LIN {X 0,Y 516.769,Z 315.126,A -85,B 0,C 180,E1 -4914.686,E2 -4914.686} C_VEL
LIN {X 0,Y 516.792,Z 318.611,A -85,B 0,C 180,E1 -4917.047,E2 -4917.047} C_VEL
LIN {X 0,Y 516.703,Z 322.745,A -85,B 0,C 180,E1 -4919.785,E2 -4919.785} C_VEL
LIN {X 0,Y 516.62,Z 326.844,A -85,B 0,C 180,E1 -4922.451,E2 -4922.451} C_VEL
LIN {X 0,Y 516.569,Z 330.921,A -85,B 0,C 180,E1 -4925.055,E2 -4925.055} C_VEL
LIN {X 0,Y 516.482,Z 335.169,A -85,B 0,C 180,E1 -4927.715,E2 -4927.715} C_VEL
LIN {X 0,Y 516.394,Z 340.454,A -85,B 0,C 180,E1 -4930.936,E2 -4930.936} C_VEL
LIN {X 0,Y 516.331,Z 344.572,A -85,B 0,C 180,E1 -4933.392,E2 -4933.392} C_VEL
LIN {X 0,Y 516.365,Z 349.185,A -85,B 0,C 180,E1 -4936.121,E2 -4936.121} C_VEL
LIN {X 0,Y 516.368,Z 349.452,A -85,B 0,C 180,E1 -4936.184,E2 -4936.184} C_VEL
LIN {X 0,Y 518.473,Z 361.595,A -85,B 0,C 180,E1 -4936.553,E2 -4936.553} C_VEL
LIN {X 0,Y 518.217,Z 374.075,A -85,B 0,C 180,E1 -4937.02,E2 -4937.02} C_VEL
LIN {X 0,Y 517.915,Z 385.417,A -85,B 0,C 180,E1 -4937.593,E2 -4937.593} C_VEL
LIN {X 0,Y 517.665,Z 396.987,A -85,B 0,C 180,E1 -4938.35,E2 -4938.35} C_VEL
LIN {X 0,Y 517.369,Z 407.679,A -85,B 0,C 180,E1 -4939.236,E2 -4939.236} C_VEL
LIN {X 0,Y 517.06,Z 417.299,A -85,B 0,C 180,E1 -4940.218,E2 -4940.218} C_VEL
LIN {X 0,Y 516.853,Z 425.177,A -85,B 0,C 180,E1 -4941.201,E2 -4941.201} C_VEL
LIN {X 0,Y 516.613,Z 432.881,A -85,B 0,C 180,E1 -4942.378,E2 -4942.378} C_VEL
LIN {X 0,Y 516.468,Z 439.944,A -85,B 0,C 180,E1 -4943.751,E2 -4943.751} C_VEL
LIN {X 0,Y 516.313,Z 444.654,A -85,B 0,C 180,E1 -4944.924,E2 -4944.924} C_VEL
LIN {X 0,Y 516.373,Z 448.256,A -85,B 0,C 180,E1 -4946.098,E2 -4946.098} C_VEL
LIN {X 0,Y 516.282,Z 450.122,A -85,B 0,C 180,E1 -4946.879,E2 -4946.879} C_VEL
LIN {X 0,Y 516.262,Z 451.529,A -85,B 0,C 180,E1 -4947.66,E2 -4947.66} C_VEL
LIN {X 0,Y 516.16,Z 453.147,A -85,B 0,C 180,E1 -4949.22,E2 -4949.22} C_VEL
LIN {X 0,Y 516.155,Z 453.384,A -85,B 0,C 180,E1 -4950,E2 -4950} C_VEL
LIN {X 0,Y 516.16,Z 453.201,A -85,B 0,C 180,E1 -4950.78,E2 -4950.78} C_VEL
LIN {X 0,Y 516.262,Z 451.653,A -85,B 0,C 180,E1 -4952.341,E2 -4952.341} C_VEL
LIN {X 0,Y 516.283,Z 450.3,A -85,B 0,C 180,E1 -4953.122,E2 -4953.122} C_VEL
LIN {X 0,Y 516.362,Z 447.439,A -85,B 0,C 180,E1 -4954.293,E2 -4954.293} C_VEL
LIN {X 0,Y 516.404,Z 443.561,A -85,B 0,C 180,E1 -4955.467,E2 -4955.467} C_VEL
LIN {X 0,Y 516.491,Z 437.713,A -85,B 0,C 180,E1 -4956.814,E2 -4956.814} C_VEL
LIN {X 0,Y 516.667,Z 431.036,A -85,B 0,C 180,E1 -4958.015,E2 -4958.015} C_VEL
LIN {X 0,Y 516.872,Z 422.892,A -85,B 0,C 180,E1 -4959.194,E2 -4959.194} C_VEL
LIN {X 0,Y 517.116,Z 414.554,A -85,B 0,C 180,E1 -4960.177,E2 -4960.177} C_VEL
LIN {X 0,Y 517.451,Z 404.26,A -85,B 0,C 180,E1 -4961.16,E2 -4961.16} C_VEL
LIN {X 0,Y 517.728,Z 393.047,A -85,B 0,C 180,E1 -4962.018,E2 -4962.018} C_VEL
LIN {X 0,Y 517.966,Z 382.905,A -85,B 0,C 180,E1 -4962.638,E2 -4962.638} C_VEL
LIN {X 0,Y 518.356,Z 370.372,A -85,B 0,C 180,E1 -4963.226,E2 -4963.226} C_VEL
LIN {X 0,Y 518.325,Z 360.107,A -85,B 0,C 180,E1 -4963.589,E2 -4963.589} C_VEL
LIN {X 0,Y 516.374,Z 349.251,A -85,B 0,C 180,E1 -4963.93,E2 -4963.93} C_VEL
LIN {X 0,Y 516.317,Z 344.726,A -85,B 0,C 180,E1 -4966.61,E2 -4966.61} C_VEL
LIN {X 0,Y 516.386,Z 340.608,A -85,B 0,C 180,E1 -4969.065,E2 -4969.065} C_VEL
LIN {X 0,Y 516.483,Z 335.316,A -85,B 0,C 180,E1 -4972.285,E2 -4972.285} C_VEL
LIN {X 0,Y 516.554,Z 331.064,A -85,B 0,C 180,E1 -4974.946,E2 -4974.946} C_VEL
LIN {X 0,Y 516.636,Z 326.528,A -85,B 0,C 180,E1 -4977.844,E2 -4977.844} C_VEL
LIN {X 0,Y 516.679,Z 322.893,A -85,B 0,C 180,E1 -4980.217,E2 -4980.217} C_VEL
LIN {X 0,Y 516.794,Z 318.755,A -85,B 0,C 180,E1 -4982.954,E2 -4982.954} C_VEL
LIN {X 0,Y 516.804,Z 315.253,A -85,B 0,C 180,E1 -4985.319,E2 -4985.319} C_VEL
LIN {X 0,Y 516.878,Z 315.1,A -85,B 0,C 180,E1 -4987.942,E2 -4987.942} C_VEL
LIN {X 0,Y 516.884,Z 315.101,A -85,B 0,C 180,E1 -4990.741,E2 -4990.741} C_VEL
LIN {X 0,Y 516.883,Z 315.098,A -85,B 0,C 180,E1 -4992.831,E2 -4992.831} C_VEL
LIN {X 0,Y 516.894,Z 315.096,A -85,B 0,C 180,E1 -4995.006,E2 -4995.006} C_VEL
LIN {X 0,Y 516.853,Z 315.103,A -85,B 0,C 180,E1 -4998.406,E2 -4998.406} C_VEL
LIN {X 0,Y 516.874,Z 315.1,A -85,B 0,C 180,E1 -5001.283,E2 -5001.283} C_VEL
LIN {X 0,Y 516.887,Z 315.101,A -85,B 0,C 180,E1 -5004.221,E2 -5004.221} C_VEL
LIN {X 0,Y 516.893,Z 315.098,A -85,B 0,C 180,E1 -5007.053,E2 -5007.053} C_VEL
LIN {X 0,Y 516.863,Z 315.1,A -85,B 0,C 180,E1 -5009.794,E2 -5009.794} C_VEL
LIN {X 0,Y 516.871,Z 315.102,A -85,B 0,C 180,E1 -5012.464,E2 -5012.464} C_VEL
LIN {X 0,Y 516.846,Z 315.104,A -85,B 0,C 180,E1 -5015.068,E2 -5015.068} C_VEL
LIN {X 0,Y 516.864,Z 315.105,A -85,B 0,C 180,E1 -5017.621,E2 -5017.621} C_VEL
LIN {X 0,Y 516.928,Z 315.093,A -85,B 0,C 180,E1 -5020.13,E2 -5020.13} C_VEL
LIN {X 0,Y 516.915,Z 315.096,A -85,B 0,C 180,E1 -5022.596,E2 -5022.596} C_VEL
LIN {X 0,Y 516.934,Z 315.093,A -85,B 0,C 180,E1 -5025.03,E2 -5025.03} C_VEL
LIN {X 0,Y 516.961,Z 315.094,A -85,B 0,C 180,E1 -5028.233,E2 -5028.233} C_VEL
LIN {X 0,Y 516.964,Z 315.092,A -85,B 0,C 180,E1 -5031.4,E2 -5031.4} C_VEL
LIN {X 0,Y 517.012,Z 315.083,A -85,B 0,C 180,E1 -5033.757,E2 -5033.757} C_VEL
LIN {X 0,Y 517.079,Z 315.073,A -85,B 0,C 180,E1 -5037.663,E2 -5037.663} C_VEL
LIN {X 0,Y 517.038,Z 315.079,A -85,B 0,C 180,E1 -5040.779,E2 -5040.779} C_VEL
LIN {X 0,Y 517.004,Z 315.086,A -85,B 0,C 180,E1 -5043.117,E2 -5043.117} C_VEL
LIN {X 0,Y 517.012,Z 315.083,A -85,B 0,C 180,E1 -5046.243,E2 -5046.243} C_VEL
LIN {X 0,Y 516.95,Z 315.089,A -85,B 0,C 180,E1 -5049.389,E2 -5049.389} C_VEL
LIN {X 0,Y 516.946,Z 315.093,A -85,B 0,C 180,E1 -5051.807,E2 -5051.807} C_VEL
LIN {X 0,Y 516.93,Z 315.094,A -85,B 0,C 180,E1 -5055.143,E2 -5055.143} C_VEL
LIN {X 0,Y 516.92,Z 315.095,A -85,B 0,C 180,E1 -5058.222,E2 -5058.222} C_VEL
LIN {X 0,Y 516.909,Z 315.098,A -85,B 0,C 180,E1 -5060.702,E2 -5060.702} C_VEL
LIN {X 0,Y 516.868,Z 315.1,A -85,B 0,C 180,E1 -5063.224,E2 -5063.224} C_VEL
LIN {X 0,Y 516.893,Z 315.097,A -85,B 0,C 180,E1 -5066.186,E2 -5066.186} C_VEL
LIN {X 0,Y 516.881,Z 315.101,A -85,B 0,C 180,E1 -5069.519,E2 -5069.519} C_VEL
LIN {X 0,Y 516.894,Z 315.1,A -85,B 0,C 180,E1 -5072.544,E2 -5072.544} C_VEL
LIN {X 0,Y 516.878,Z 315.1,A -85,B 0,C 180,E1 -5075.332,E2 -5075.332} C_VEL
LIN {X 0,Y 516.877,Z 315.101,A -85,B 0,C 180,E1 -5077.943,E2 -5077.943} C_VEL
LIN {X 0,Y 516.849,Z 315.103,A -85,B 0,C 180,E1 -5080.745,E2 -5080.745} C_VEL
LIN {X 0,Y 516.878,Z 315.099,A -85,B 0,C 180,E1 -5083.904,E2 -5083.904} C_VEL
LIN {X 0,Y 516.88,Z 315.103,A -85,B 0,C 180,E1 -5086.107,E2 -5086.107} C_VEL
LIN {X 0,Y 516.915,Z 315.097,A -85,B 0,C 180,E1 -5088.399,E2 -5088.399} C_VEL
LIN {X 0,Y 516.88,Z 315.104,A -85,B 0,C 180,E1 -5091.284,E2 -5091.284} C_VEL
LIN {X 0,Y 516.893,Z 315.205,A -85,B 0,C 180,E1 -5092.277,E2 -5092.277} C_VEL
LIN {X 0,Y 517.584,Z 320.371,A -85,B 0,C 180,E1 -5094.559,E2 -5094.559} C_VEL
LIN {X 0,Y 517.453,Z 327.148,A -85,B 0,C 180,E1 -5097.361,E2 -5097.361} C_VEL
LIN {X 0,Y 517.277,Z 334.775,A -85,B 0,C 180,E1 -5100.405,E2 -5100.405} C_VEL
LIN {X 0,Y 517.083,Z 342.335,A -85,B 0,C 180,E1 -5103.351,E2 -5103.351} C_VEL
LIN {X 0,Y 516.938,Z 350.126,A -85,B 0,C 180,E1 -5106.355,E2 -5106.355} C_VEL
LIN {X 0,Y 516.789,Z 357.918,A -85,B 0,C 180,E1 -5109.293,E2 -5109.293} C_VEL
LIN {X 0,Y 516.635,Z 365.829,A -85,B 0,C 180,E1 -5112.221,E2 -5112.221} C_VEL
LIN {X 0,Y 516.567,Z 373.5,A -85,B 0,C 180,E1 -5115.019,E2 -5115.019} C_VEL
LIN {X 0,Y 516.505,Z 376.491,A -85,B 0,C 180,E1 -5116.099,E2 -5116.099} C_VEL
LIN {X 0,Y 518.478,Z 389.092,A -85,B 0,C 180,E1 -5116.453,E2 -5116.453} C_VEL
LIN {X 0,Y 518.244,Z 402.111,A -85,B 0,C 180,E1 -5116.92,E2 -5116.92} C_VEL
LIN {X 0,Y 517.912,Z 414.402,A -85,B 0,C 180,E1 -5117.529,E2 -5117.529} C_VEL
LIN {X 0,Y 517.617,Z 425.586,A -85,B 0,C 180,E1 -5118.249,E2 -5118.249} C_VEL
LIN {X 0,Y 517.328,Z 436.469,A -85,B 0,C 180,E1 -5119.135,E2 -5119.135} C_VEL
LIN {X 0,Y 517.044,Z 445.333,A -85,B 0,C 180,E1 -5120.02,E2 -5120.02} C_VEL
LIN {X 0,Y 516.814,Z 454.959,A -85,B 0,C 180,E1 -5121.2,E2 -5121.2} C_VEL
LIN {X 0,Y 516.563,Z 462.62,A -85,B 0,C 180,E1 -5122.377,E2 -5122.377} C_VEL
LIN {X 0,Y 516.427,Z 469.679,A -85,B 0,C 180,E1 -5123.75,E2 -5123.75} C_VEL
LIN {X 0,Y 516.313,Z 474.372,A -85,B 0,C 180,E1 -5124.924,E2 -5124.924} C_VEL
LIN {X 0,Y 516.355,Z 477.957,A -85,B 0,C 180,E1 -5126.098,E2 -5126.098} C_VEL
LIN {X 0,Y 516.282,Z 479.807,A -85,B 0,C 180,E1 -5126.878,E2 -5126.878} C_VEL
LIN {X 0,Y 516.261,Z 481.196,A -85,B 0,C 180,E1 -5127.659,E2 -5127.659} C_VEL
LIN {X 0,Y 516.16,Z 482.785,A -85,B 0,C 180,E1 -5129.22,E2 -5129.22} C_VEL
LIN {X 0,Y 516.154,Z 483,A -85,B 0,C 180,E1 -5130,E2 -5130} C_VEL
LIN {X 0,Y 516.192,Z 482.186,A -85,B 0,C 180,E1 -5131.56,E2 -5131.56} C_VEL
LIN {X 0,Y 516.261,Z 481.199,A -85,B 0,C 180,E1 -5132.34,E2 -5132.34} C_VEL
LIN {X 0,Y 516.282,Z 479.811,A -85,B 0,C 180,E1 -5133.121,E2 -5133.121} C_VEL
LIN {X 0,Y 516.343,Z 476.897,A -85,B 0,C 180,E1 -5134.293,E2 -5134.293} C_VEL
LIN {X 0,Y 516.405,Z 472.95,A -85,B 0,C 180,E1 -5135.466,E2 -5135.466} C_VEL
LIN {X 0,Y 516.485,Z 467.035,A -85,B 0,C 180,E1 -5136.807,E2 -5136.807} C_VEL
LIN {X 0,Y 516.64,Z 460.24,A -85,B 0,C 180,E1 -5138.015,E2 -5138.015} C_VEL
LIN {X 0,Y 516.867,Z 451.995,A -85,B 0,C 180,E1 -5139.193,E2 -5139.193} C_VEL
LIN {X 0,Y 517.08,Z 443.544,A -85,B 0,C 180,E1 -5140.177,E2 -5140.177} C_VEL
LIN {X 0,Y 517.46,Z 433.103,A -85,B 0,C 180,E1 -5141.159,E2 -5141.159} C_VEL
LIN {X 0,Y 517.696,Z 421.809,A -85,B 0,C 180,E1 -5142.014,E2 -5142.014} C_VEL
LIN {X 0,Y 517.97,Z 411.419,A -85,B 0,C 180,E1 -5142.637,E2 -5142.637} C_VEL
LIN {X 0,Y 518.28,Z 399.779,A -85,B 0,C 180,E1 -5143.178,E2 -5143.178} C_VEL
LIN {X 0,Y 518.314,Z 387.284,A -85,B 0,C 180,E1 -5143.601,E2 -5143.601} C_VEL
LIN {X 0,Y 516.504,Z 376.493,A -85,B 0,C 180,E1 -5143.9,E2 -5143.9} C_VEL
LIN {X 0,Y 516.576,Z 369.05,A -85,B 0,C 180,E1 -5146.6,E2 -5146.6} C_VEL
LIN {X 0,Y 516.77,Z 360.146,A -85,B 0,C 180,E1 -5149.876,E2 -5149.876} C_VEL
LIN {X 0,Y 516.909,Z 352.356,A -85,B 0,C 180,E1 -5152.797,E2 -5152.797} C_VEL
LIN {X 0,Y 517.036,Z 344.563,A -85,B 0,C 180,E1 -5155.783,E2 -5155.783} C_VEL
LIN {X 0,Y 517.178,Z 337.818,A -85,B 0,C 180,E1 -5158.399,E2 -5158.399} C_VEL
LIN {X 0,Y 517.364,Z 330.793,A -85,B 0,C 180,E1 -5161.151,E2 -5161.151} C_VEL
LIN {X 0,Y 517.541,Z 323.649,A -85,B 0,C 180,E1 -5164.07,E2 -5164.07} C_VEL
LIN {X 0,Y 517.565,Z 319.707,A -85,B 0,C 180,E1 -5165.724,E2 -5165.724} C_VEL
LIN {X 0,Y 516.89,Z 315.102,A -85,B 0,C 180,E1 -5167.8,E2 -5167.8} C_VEL
LIN {X 0,Y 516.9,Z 315.1,A -85,B 0,C 180,E1 -5170.739,E2 -5170.739} C_VEL
LIN {X 0,Y 516.878,Z 315.105,A -85,B 0,C 180,E1 -5173.902,E2 -5173.902} C_VEL
LIN {X 0,Y 516.875,Z 315.099,A -85,B 0,C 180,E1 -5176.106,E2 -5176.106} C_VEL
LIN {X 0,Y 516.853,Z 315.102,A -85,B 0,C 180,E1 -5179.255,E2 -5179.255} C_VEL
LIN {X 0,Y 516.873,Z 315.101,A -85,B 0,C 180,E1 -5182.056,E2 -5182.056} C_VEL
LIN {X 0,Y 516.887,Z 315.099,A -85,B 0,C 180,E1 -5185.175,E2 -5185.175} C_VEL
LIN {X 0,Y 516.867,Z 315.102,A -85,B 0,C 180,E1 -5187.975,E2 -5187.975} C_VEL
LIN {X 0,Y 516.893,Z 315.102,A -85,B 0,C 180,E1 -5190.694,E2 -5190.694} C_VEL
LIN {X 0,Y 516.893,Z 315.097,A -85,B 0,C 180,E1 -5193.812,E2 -5193.812} C_VEL
LIN {X 0,Y 516.862,Z 315.101,A -85,B 0,C 180,E1 -5196.776,E2 -5196.776} C_VEL
LIN {X 0,Y 516.93,Z 315.096,A -85,B 0,C 180,E1 -5199.731,E2 -5199.731} C_VEL
LIN {X 0,Y 516.916,Z 315.098,A -85,B 0,C 180,E1 -5202.596,E2 -5202.596} C_VEL
LIN {X 0,Y 516.923,Z 315.094,A -85,B 0,C 180,E1 -5205.03,E2 -5205.03} C_VEL
LIN {X 0,Y 516.955,Z 315.092,A -85,B 0,C 180,E1 -5208.233,E2 -5208.233} C_VEL
LIN {X 0,Y 516.962,Z 315.092,A -85,B 0,C 180,E1 -5211.4,E2 -5211.4} C_VEL
LIN {X 0,Y 517.053,Z 315.08,A -85,B 0,C 180,E1 -5214.54,E2 -5214.54} C_VEL
LIN {X 0,Y 517.074,Z 315.075,A -85,B 0,C 180,E1 -5217.663,E2 -5217.663} C_VEL
LIN {X 0,Y 517.053,Z 315.076,A -85,B 0,C 180,E1 -5220.779,E2 -5220.779} C_VEL
LIN {X 0,Y 517.001,Z 315.085,A -85,B 0,C 180,E1 -5223.117,E2 -5223.117} C_VEL
LIN {X 0,Y 517.007,Z 315.083,A -85,B 0,C 180,E1 -5226.243,E2 -5226.243} C_VEL
LIN {X 0,Y 516.946,Z 315.091,A -85,B 0,C 180,E1 -5229.389,E2 -5229.389} C_VEL
LIN {X 0,Y 516.94,Z 315.096,A -85,B 0,C 180,E1 -5231.807,E2 -5231.807} C_VEL
LIN {X 0,Y 516.927,Z 315.095,A -85,B 0,C 180,E1 -5235.144,E2 -5235.144} C_VEL
LIN {X 0,Y 516.916,Z 315.094,A -85,B 0,C 180,E1 -5238.223,E2 -5238.223} C_VEL
LIN {X 0,Y 516.904,Z 315.101,A -85,B 0,C 180,E1 -5240.702,E2 -5240.702} C_VEL
LIN {X 0,Y 516.863,Z 315.101,A -85,B 0,C 180,E1 -5243.224,E2 -5243.224} C_VEL
LIN {X 0,Y 516.893,Z 315.099,A -85,B 0,C 180,E1 -5246.188,E2 -5246.188} C_VEL
LIN {X 0,Y 516.876,Z 315.1,A -85,B 0,C 180,E1 -5249.519,E2 -5249.519} C_VEL
LIN {X 0,Y 516.89,Z 315.102,A -85,B 0,C 180,E1 -5252.545,E2 -5252.545} C_VEL
LIN {X 0,Y 516.876,Z 315.1,A -85,B 0,C 180,E1 -5255.333,E2 -5255.333} C_VEL
LIN {X 0,Y 516.873,Z 315.103,A -85,B 0,C 180,E1 -5257.944,E2 -5257.944} C_VEL
LIN {X 0,Y 516.854,Z 315.104,A -85,B 0,C 180,E1 -5260.745,E2 -5260.745} C_VEL
LIN {X 0,Y 516.875,Z 315.099,A -85,B 0,C 180,E1 -5263.904,E2 -5263.904} C_VEL
LIN {X 0,Y 516.863,Z 315.099,A -85,B 0,C 180,E1 -5266.924,E2 -5266.924} C_VEL
LIN {X 0,Y 516.905,Z 315.098,A -85,B 0,C 180,E1 -5269.588,E2 -5269.588} C_VEL
LIN {X 0,Y 516.898,Z 315.097,A -85,B 0,C 180,E1 -5270.31,E2 -5270.31} C_VEL
LIN {X 0,Y 516.218,Z 315.184,A -85,B 0,C 180,E1 -5270.96,E2 -5270.96} C_VEL
LIN {X 0,Y 513.359,Z 315.539,A -85,B 0,C 180,E1 -5272.015,E2 -5272.015} C_VEL
LIN {X 0,Y 510.934,Z 315.843,A -85,B 0,C 180,E1 -5272.865,E2 -5272.865} C_VEL
LIN {X 0,Y 509.869,Z 315.975,A -85,B 0,C 180,E1 -5273.522,E2 -5273.522} C_VEL
LIN {X 0,Y 509.769,Z 315.986,A -85,B 0,C 180,E1 -5273.744,E2 -5273.744} C_VEL
LIN {X 0,Y 509.741,Z 315.993,A -85,B 0,C 180,E1 -5274.616,E2 -5274.616} C_VEL
LIN {X 0,Y 509.762,Z 318.703,A -85,B 0,C 180,E1 -5276.533,E2 -5276.533} C_VEL
LIN {X 0,Y 509.647,Z 322.848,A -85,B 0,C 180,E1 -5279.322,E2 -5279.322} C_VEL
LIN {X 0,Y 509.592,Z 326.962,A -85,B 0,C 180,E1 -5282.038,E2 -5282.038} C_VEL
LIN {X 0,Y 509.535,Z 332.407,A -85,B 0,C 180,E1 -5285.558,E2 -5285.558} C_VEL
LIN {X 0,Y 509.372,Z 336.479,A -85,B 0,C 180,E1 -5288.129,E2 -5288.129} C_VEL
LIN {X 0,Y 509.318,Z 340.577,A -85,B 0,C 180,E1 -5290.661,E2 -5290.661} C_VEL
LIN {X 0,Y 509.269,Z 344.729,A -85,B 0,C 180,E1 -5293.155,E2 -5293.155} C_VEL
LIN {X 0,Y 509.311,Z 349.492,A -85,B 0,C 180,E1 -5295.976,E2 -5295.976} C_VEL
LIN {X 0,Y 511.573,Z 362.589,A -85,B 0,C 180,E1 -5296.393,E2 -5296.393} C_VEL
LIN {X 0,Y 511.276,Z 375.432,A -85,B 0,C 180,E1 -5296.891,E2 -5296.891} C_VEL
LIN {X 0,Y 510.976,Z 387.064,A -85,B 0,C 180,E1 -5297.504,E2 -5297.504} C_VEL
LIN {X 0,Y 510.698,Z 398.496,A -85,B 0,C 180,E1 -5298.289,E2 -5298.289} C_VEL
LIN {X 0,Y 510.363,Z 408.966,A -85,B 0,C 180,E1 -5299.186,E2 -5299.186} C_VEL
LIN {X 0,Y 510.066,Z 417.52,A -85,B 0,C 180,E1 -5300.083,E2 -5300.083} C_VEL
LIN {X 0,Y 509.836,Z 425.397,A -85,B 0,C 180,E1 -5301.079,E2 -5301.079} C_VEL
LIN {X 0,Y 509.569,Z 433.1,A -85,B 0,C 180,E1 -5302.272,E2 -5302.272} C_VEL
LIN {X 0,Y 509.403,Z 440.162,A -85,B 0,C 180,E1 -5303.664,E2 -5303.664} C_VEL
LIN {X 0,Y 509.248,Z 444.871,A -85,B 0,C 180,E1 -5304.854,E2 -5304.854} C_VEL
LIN {X 0,Y 509.303,Z 448.473,A -85,B 0,C 180,E1 -5306.044,E2 -5306.044} C_VEL
LIN {X 0,Y 509.201,Z 450.339,A -85,B 0,C 180,E1 -5306.836,E2 -5306.836} C_VEL
LIN {X 0,Y 509.19,Z 451.744,A -85,B 0,C 180,E1 -5307.627,E2 -5307.627} C_VEL
LIN {X 0,Y 509.074,Z 453.362,A -85,B 0,C 180,E1 -5309.209,E2 -5309.209} C_VEL
LIN {X 0,Y 509.066,Z 453.599,A -85,B 0,C 180,E1 -5310,E2 -5310} C_VEL
LIN {X 0,Y 509.074,Z 453.416,A -85,B 0,C 180,E1 -5310.791,E2 -5310.791} C_VEL
LIN {X 0,Y 509.19,Z 451.867,A -85,B 0,C 180,E1 -5312.373,E2 -5312.373} C_VEL
LIN {X 0,Y 509.202,Z 450.514,A -85,B 0,C 180,E1 -5313.165,E2 -5313.165} C_VEL
LIN {X 0,Y 509.284,Z 447.653,A -85,B 0,C 180,E1 -5314.353,E2 -5314.353} C_VEL
LIN {X 0,Y 509.347,Z 443.774,A -85,B 0,C 180,E1 -5315.543,E2 -5315.543} C_VEL
LIN {X 0,Y 509.419,Z 438.149,A -85,B 0,C 180,E1 -5316.865,E2 -5316.865} C_VEL
LIN {X 0,Y 509.63,Z 431.248,A -85,B 0,C 180,E1 -5318.126,E2 -5318.126} C_VEL
LIN {X 0,Y 509.86,Z 423.103,A -85,B 0,C 180,E1 -5319.321,E2 -5319.321} C_VEL
LIN {X 0,Y 510.118,Z 414.765,A -85,B 0,C 180,E1 -5320.318,E2 -5320.318} C_VEL
LIN {X 0,Y 510.498,Z 404.467,A -85,B 0,C 180,E1 -5321.314,E2 -5321.314} C_VEL
LIN {X 0,Y 510.781,Z 393.254,A -85,B 0,C 180,E1 -5322.184,E2 -5322.184} C_VEL
LIN {X 0,Y 511.038,Z 383.11,A -85,B 0,C 180,E1 -5322.812,E2 -5322.812} C_VEL
LIN {X 0,Y 511.466,Z 370.571,A -85,B 0,C 180,E1 -5323.408,E2 -5323.408} C_VEL
LIN {X 0,Y 511.377,Z 360.716,A -85,B 0,C 180,E1 -5323.765,E2 -5323.765} C_VEL
LIN {X 0,Y 509.3,Z 349.471,A -85,B 0,C 180,E1 -5324.127,E2 -5324.127} C_VEL
LIN {X 0,Y 509.255,Z 344.881,A -85,B 0,C 180,E1 -5326.847,E2 -5326.847} C_VEL
LIN {X 0,Y 509.313,Z 340.73,A -85,B 0,C 180,E1 -5329.34,E2 -5329.34} C_VEL
LIN {X 0,Y 509.425,Z 335.728,A -85,B 0,C 180,E1 -5332.432,E2 -5332.432} C_VEL
LIN {X 0,Y 509.492,Z 331.193,A -85,B 0,C 180,E1 -5335.316,E2 -5335.316} C_VEL
LIN {X 0,Y 509.572,Z 327,A -85,B 0,C 180,E1 -5338.031,E2 -5338.031} C_VEL
LIN {X 0,Y 509.655,Z 322.148,A -85,B 0,C 180,E1 -5341.244,E2 -5341.244} C_VEL
LIN {X 0,Y 509.812,Z 317.769,A -85,B 0,C 180,E1 -5344.195,E2 -5344.195} C_VEL
LIN {X 0,Y 509.767,Z 315.987,A -85,B 0,C 180,E1 -5345.569,E2 -5345.569} C_VEL
LIN {X 0,Y 509.848,Z 315.978,A -85,B 0,C 180,E1 -5348.338,E2 -5348.338} C_VEL
LIN {X 0,Y 509.857,Z 315.974,A -85,B 0,C 180,E1 -5351.425,E2 -5351.425} C_VEL
LIN {X 0,Y 509.838,Z 315.974,A -85,B 0,C 180,E1 -5354.669,E2 -5354.669} C_VEL
LIN {X 0,Y 509.789,Z 315.985,A -85,B 0,C 180,E1 -5357.505,E2 -5357.505} C_VEL
LIN {X 0,Y 509.83,Z 315.98,A -85,B 0,C 180,E1 -5360.646,E2 -5360.646} C_VEL
LIN {X 0,Y 509.832,Z 315.979,A -85,B 0,C 180,E1 -5363.647,E2 -5363.647} C_VEL
LIN {X 0,Y 509.859,Z 315.973,A -85,B 0,C 180,E1 -5366.539,E2 -5366.539} C_VEL
LIN {X 0,Y 509.831,Z 315.981,A -85,B 0,C 180,E1 -5369.333,E2 -5369.333} C_VEL
LIN {X 0,Y 509.827,Z 315.977,A -85,B 0,C 180,E1 -5372.05,E2 -5372.05} C_VEL
LIN {X 0,Y 509.802,Z 315.983,A -85,B 0,C 180,E1 -5374.7,E2 -5374.7} C_VEL
LIN {X 0,Y 509.822,Z 315.981,A -85,B 0,C 180,E1 -5377.458,E2 -5377.458} C_VEL
LIN {X 0,Y 509.913,Z 315.968,A -85,B 0,C 180,E1 -5379.844,E2 -5379.844} C_VEL
LIN {X 0,Y 509.874,Z 315.973,A -85,B 0,C 180,E1 -5383.174,E2 -5383.174} C_VEL
LIN {X 0,Y 509.847,Z 315.974,A -85,B 0,C 180,E1 -5385.634,E2 -5385.634} C_VEL
LIN {X 0,Y 509.907,Z 315.968,A -85,B 0,C 180,E1 -5388.874,E2 -5388.874} C_VEL
LIN {X 0,Y 509.947,Z 315.964,A -85,B 0,C 180,E1 -5392.078,E2 -5392.078} C_VEL
LIN {X 0,Y 509.982,Z 315.96,A -85,B 0,C 180,E1 -5394.464,E2 -5394.464} C_VEL
LIN {X 0,Y 510.049,Z 315.948,A -85,B 0,C 180,E1 -5397.631,E2 -5397.631} C_VEL
LIN {X 0,Y 509.99,Z 315.957,A -85,B 0,C 180,E1 -5400.79,E2 -5400.79} C_VEL
LIN {X 0,Y 509.946,Z 315.965,A -85,B 0,C 180,E1 -5403.16,E2 -5403.16} C_VEL
LIN {X 0,Y 509.979,Z 315.96,A -85,B 0,C 180,E1 -5406.33,E2 -5406.33} C_VEL
LIN {X 0,Y 509.913,Z 315.969,A -85,B 0,C 180,E1 -5408.72,E2 -5408.72} C_VEL
LIN {X 0,Y 509.898,Z 315.973,A -85,B 0,C 180,E1 -5411.932,E2 -5411.932} C_VEL
LIN {X 0,Y 509.889,Z 315.972,A -85,B 0,C 180,E1 -5415.242,E2 -5415.242} C_VEL
LIN {X 0,Y 509.862,Z 315.976,A -85,B 0,C 180,E1 -5418.484,E2 -5418.484} C_VEL
LIN {X 0,Y 509.847,Z 315.977,A -85,B 0,C 180,E1 -5421.002,E2 -5421.002} C_VEL
LIN {X 0,Y 509.826,Z 315.979,A -85,B 0,C 180,E1 -5423.564,E2 -5423.564} C_VEL
LIN {X 0,Y 509.849,Z 315.973,A -85,B 0,C 180,E1 -5426.366,E2 -5426.366} C_VEL
LIN {X 0,Y 509.848,Z 315.975,A -85,B 0,C 180,E1 -5429.725,E2 -5429.725} C_VEL
LIN {X 0,Y 509.871,Z 315.976,A -85,B 0,C 180,E1 -5432.775,E2 -5432.775} C_VEL
LIN {X 0,Y 509.838,Z 315.978,A -85,B 0,C 180,E1 -5435.581,E2 -5435.581} C_VEL
LIN {X 0,Y 509.846,Z 315.975,A -85,B 0,C 180,E1 -5438.339,E2 -5438.339} C_VEL
LIN {X 0,Y 509.804,Z 315.982,A -85,B 0,C 180,E1 -5441.431,E2 -5441.431} C_VEL
LIN {X 0,Y 509.837,Z 315.981,A -85,B 0,C 180,E1 -5444.67,E2 -5444.67} C_VEL
LIN {X 0,Y 509.857,Z 315.979,A -85,B 0,C 180,E1 -5448.104,E2 -5448.104} C_VEL
LIN {X 0,Y 509.845,Z 315.978,A -85,B 0,C 180,E1 -5450.648,E2 -5450.648} C_VEL
LIN {X 0,Y 509.881,Z 316.03,A -85,B 0,C 180,E1 -5452.072,E2 -5452.072} C_VEL
LIN {X 0,Y 510.556,Z 320.994,A -85,B 0,C 180,E1 -5454.308,E2 -5454.308} C_VEL
LIN {X 0,Y 510.523,Z 326.406,A -85,B 0,C 180,E1 -5456.589,E2 -5456.589} C_VEL
LIN {X 0,Y 510.308,Z 333.217,A -85,B 0,C 180,E1 -5459.365,E2 -5459.365} C_VEL
LIN {X 0,Y 510.169,Z 340.015,A -85,B 0,C 180,E1 -5462.071,E2 -5462.071} C_VEL
LIN {X 0,Y 510,Z 346.787,A -85,B 0,C 180,E1 -5464.711,E2 -5464.711} C_VEL
LIN {X 0,Y 509.854,Z 353.867,A -85,B 0,C 180,E1 -5467.451,E2 -5467.451} C_VEL
LIN {X 0,Y 509.654,Z 362.37,A -85,B 0,C 180,E1 -5470.673,E2 -5470.673} C_VEL
LIN {X 0,Y 509.517,Z 371.274,A -85,B 0,C 180,E1 -5473.986,E2 -5473.986} C_VEL
LIN {X 0,Y 509.444,Z 376.491,A -85,B 0,C 180,E1 -5475.902,E2 -5475.902} C_VEL
LIN {X 0,Y 511.563,Z 389.927,A -85,B 0,C 180,E1 -5476.291,E2 -5476.291} C_VEL
LIN {X 0,Y 511.342,Z 402.11,A -85,B 0,C 180,E1 -5476.741,E2 -5476.741} C_VEL
LIN {X 0,Y 510.992,Z 413.172,A -85,B 0,C 180,E1 -5477.287,E2 -5477.287} C_VEL
LIN {X 0,Y 510.741,Z 423.844,A -85,B 0,C 180,E1 -5477.964,E2 -5477.964} C_VEL
LIN {X 0,Y 510.429,Z 434.261,A -85,B 0,C 180,E1 -5478.785,E2 -5478.785} C_VEL
LIN {X 0,Y 510.07,Z 443.538,A -85,B 0,C 180,E1 -5479.681,E2 -5479.681} C_VEL
LIN {X 0,Y 509.846,Z 451.99,A -85,B 0,C 180,E1 -5480.679,E2 -5480.679} C_VEL
LIN {X 0,Y 509.585,Z 460.235,A -85,B 0,C 180,E1 -5481.873,E2 -5481.873} C_VEL
LIN {X 0,Y 509.419,Z 466.876,A -85,B 0,C 180,E1 -5483.067,E2 -5483.067} C_VEL
LIN {X 0,Y 509.344,Z 472.949,A -85,B 0,C 180,E1 -5484.457,E2 -5484.457} C_VEL
LIN {X 0,Y 509.234,Z 476.894,A -85,B 0,C 180,E1 -5485.646,E2 -5485.646} C_VEL
LIN {X 0,Y 509.201,Z 479.807,A -85,B 0,C 180,E1 -5486.835,E2 -5486.835} C_VEL
LIN {X 0,Y 509.161,Z 481.195,A -85,B 0,C 180,E1 -5487.626,E2 -5487.626} C_VEL
LIN {X 0,Y 509.073,Z 482.785,A -85,B 0,C 180,E1 -5489.209,E2 -5489.209} C_VEL
LIN {X 0,Y 509.065,Z 483,A -85,B 0,C 180,E1 -5490,E2 -5490} C_VEL
LIN {X 0,Y 509.112,Z 482.185,A -85,B 0,C 180,E1 -5491.582,E2 -5491.582} C_VEL
LIN {X 0,Y 509.161,Z 481.198,A -85,B 0,C 180,E1 -5492.373,E2 -5492.373} C_VEL
LIN {X 0,Y 509.2,Z 479.811,A -85,B 0,C 180,E1 -5493.164,E2 -5493.164} C_VEL
LIN {X 0,Y 509.234,Z 476.897,A -85,B 0,C 180,E1 -5494.353,E2 -5494.353} C_VEL
LIN {X 0,Y 509.344,Z 472.95,A -85,B 0,C 180,E1 -5495.542,E2 -5495.542} C_VEL
LIN {X 0,Y 509.409,Z 467.284,A -85,B 0,C 180,E1 -5496.853,E2 -5496.853} C_VEL
LIN {X 0,Y 509.584,Z 460.24,A -85,B 0,C 180,E1 -5498.126,E2 -5498.126} C_VEL
LIN {X 0,Y 509.845,Z 451.995,A -85,B 0,C 180,E1 -5499.321,E2 -5499.321} C_VEL
LIN {X 0,Y 510.069,Z 443.544,A -85,B 0,C 180,E1 -5500.318,E2 -5500.318} C_VEL
LIN {X 0,Y 510.486,Z 433.102,A -85,B 0,C 180,E1 -5501.313,E2 -5501.313} C_VEL
LIN {X 0,Y 510.729,Z 422.539,A -85,B 0,C 180,E1 -5502.129,E2 -5502.129} C_VEL
LIN {X 0,Y 511.037,Z 411.418,A -85,B 0,C 180,E1 -5502.812,E2 -5502.812} C_VEL
LIN {X 0,Y 511.374,Z 399.779,A -85,B 0,C 180,E1 -5503.359,E2 -5503.359} C_VEL
LIN {X 0,Y 511.411,Z 388.198,A -85,B 0,C 180,E1 -5503.763,E2 -5503.763} C_VEL
LIN {X 0,Y 509.443,Z 376.493,A -85,B 0,C 180,E1 -5504.097,E2 -5504.097} C_VEL
LIN {X 0,Y 509.522,Z 369.05,A -85,B 0,C 180,E1 -5506.837,E2 -5506.837} C_VEL
LIN {X 0,Y 509.711,Z 361.259,A -85,B 0,C 180,E1 -5509.743,E2 -5509.743} C_VEL
LIN {X 0,Y 509.85,Z 353.467,A -85,B 0,C 180,E1 -5512.703,E2 -5512.703} C_VEL
LIN {X 0,Y 510.001,Z 345.67,A -85,B 0,C 180,E1 -5515.726,E2 -5515.726} C_VEL
LIN {X 0,Y 510.18,Z 337.71,A -85,B 0,C 180,E1 -5518.824,E2 -5518.824} C_VEL
LIN {X 0,Y 510.375,Z 330.88,A -85,B 0,C 180,E1 -5521.551,E2 -5521.551} C_VEL
LIN {X 0,Y 510.547,Z 324.131,A -85,B 0,C 180,E1 -5524.359,E2 -5524.359} C_VEL
LIN {X 0,Y 510.453,Z 319.611,A -85,B 0,C 180,E1 -5526.3,E2 -5526.3} C_VEL
LIN {X 0,Y 509.861,Z 315.978,A -85,B 0,C 180,E1 -5528.024,E2 -5528.024} C_VEL
LIN {X 0,Y 509.855,Z 315.978,A -85,B 0,C 180,E1 -5530.7,E2 -5530.7} C_VEL
LIN {X 0,Y 509.821,Z 315.985,A -85,B 0,C 180,E1 -5533.57,E2 -5533.57} C_VEL
LIN {X 0,Y 509.803,Z 315.98,A -85,B 0,C 180,E1 -5536.426,E2 -5536.426} C_VEL
LIN {X 0,Y 509.814,Z 315.979,A -85,B 0,C 180,E1 -5539.304,E2 -5539.304} C_VEL
LIN {X 0,Y 509.843,Z 315.976,A -85,B 0,C 180,E1 -5541.786,E2 -5541.786} C_VEL
LIN {X 0,Y 509.839,Z 315.977,A -85,B 0,C 180,E1 -5544.622,E2 -5544.622} C_VEL
LIN {X 0,Y 509.855,Z 315.977,A -85,B 0,C 180,E1 -5547.48,E2 -5547.48} C_VEL
LIN {X 0,Y 509.843,Z 315.976,A -85,B 0,C 180,E1 -5550.274,E2 -5550.274} C_VEL
LIN {X 0,Y 509.868,Z 315.971,A -85,B 0,C 180,E1 -5553.629,E2 -5553.629} C_VEL
LIN {X 0,Y 509.821,Z 315.98,A -85,B 0,C 180,E1 -5556.436,E2 -5556.436} C_VEL
LIN {X 0,Y 509.907,Z 315.97,A -85,B 0,C 180,E1 -5559.844,E2 -5559.844} C_VEL
LIN {X 0,Y 509.869,Z 315.974,A -85,B 0,C 180,E1 -5563.174,E2 -5563.174} C_VEL
LIN {X 0,Y 509.841,Z 315.975,A -85,B 0,C 180,E1 -5565.633,E2 -5565.633} C_VEL
LIN {X 0,Y 509.902,Z 315.966,A -85,B 0,C 180,E1 -5568.874,E2 -5568.874} C_VEL
LIN {X 0,Y 509.942,Z 315.964,A -85,B 0,C 180,E1 -5572.078,E2 -5572.078} C_VEL
LIN {X 0,Y 510.001,Z 315.958,A -85,B 0,C 180,E1 -5574.465,E2 -5574.465} C_VEL
LIN {X 0,Y 510.045,Z 315.951,A -85,B 0,C 180,E1 -5577.631,E2 -5577.631} C_VEL
LIN {X 0,Y 510.005,Z 315.954,A -85,B 0,C 180,E1 -5580.79,E2 -5580.79} C_VEL
LIN {X 0,Y 509.944,Z 315.964,A -85,B 0,C 180,E1 -5583.16,E2 -5583.16} C_VEL
LIN {X 0,Y 509.974,Z 315.96,A -85,B 0,C 180,E1 -5586.33,E2 -5586.33} C_VEL
LIN {X 0,Y 509.908,Z 315.971,A -85,B 0,C 180,E1 -5588.72,E2 -5588.72} C_VEL
LIN {X 0,Y 509.893,Z 315.973,A -85,B 0,C 180,E1 -5591.932,E2 -5591.932} C_VEL
LIN {X 0,Y 509.883,Z 315.974,A -85,B 0,C 180,E1 -5595.242,E2 -5595.242} C_VEL
LIN {X 0,Y 509.879,Z 315.97,A -85,B 0,C 180,E1 -5598.002,E2 -5598.002} C_VEL
LIN {X 0,Y 509.842,Z 315.978,A -85,B 0,C 180,E1 -5601.002,E2 -5601.002} C_VEL
LIN {X 0,Y 509.821,Z 315.98,A -85,B 0,C 180,E1 -5603.564,E2 -5603.564} C_VEL
LIN {X 0,Y 509.868,Z 315.973,A -85,B 0,C 180,E1 -5606.371,E2 -5606.371} C_VEL
LIN {X 0,Y 509.842,Z 315.974,A -85,B 0,C 180,E1 -5609.752,E2 -5609.752} C_VEL
LIN {X 0,Y 509.867,Z 315.976,A -85,B 0,C 180,E1 -5612.775,E2 -5612.775} C_VEL
LIN {X 0,Y 509.835,Z 315.978,A -85,B 0,C 180,E1 -5615.582,E2 -5615.582} C_VEL
LIN {X 0,Y 509.843,Z 315.976,A -85,B 0,C 180,E1 -5618.339,E2 -5618.339} C_VEL
LIN {X 0,Y 509.825,Z 315.979,A -85,B 0,C 180,E1 -5621.429,E2 -5621.429} C_VEL
LIN {X 0,Y 509.833,Z 315.98,A -85,B 0,C 180,E1 -5624.671,E2 -5624.671} C_VEL
LIN {X 0,Y 509.857,Z 315.979,A -85,B 0,C 180,E1 -5628.104,E2 -5628.104} C_VEL
LIN {X 0,Y 509.856,Z 315.974,A -85,B 0,C 180,E1 -5630.65,E2 -5630.65} C_VEL
LIN {X 0,Y 509.769,Z 315.986,A -85,B 0,C 180,E1 -5633.744,E2 -5633.744} C_VEL
LIN {X 0,Y 509.069,Z 316.267,A -85,B 0,C 180,E1 -5634.402,E2 -5634.402} C_VEL
LIN {X 0,Y 506.222,Z 317.612,A -85,B 0,C 180,E1 -5635.464,E2 -5635.464} C_VEL
LIN {X 0,Y 503.822,Z 319.106,A -85,B 0,C 180,E1 -5636.315,E2 -5636.315} C_VEL
LIN {X 0,Y 502.777,Z 320.193,A -85,B 0,C 180,E1 -5636.972,E2 -5636.972} C_VEL
LIN {X 0,Y 502.683,Z 320.528,A -85,B 0,C 180,E1 -5637.195,E2 -5637.195} C_VEL
LIN {X 0,Y 502.571,Z 324.835,A -85,B 0,C 180,E1 -5640.114,E2 -5640.114} C_VEL
LIN {X 0,Y 502.486,Z 328.446,A -85,B 0,C 180,E1 -5642.514,E2 -5642.514} C_VEL
LIN {X 0,Y 502.476,Z 332.84,A -85,B 0,C 180,E1 -5645.387,E2 -5645.387} C_VEL
LIN {X 0,Y 502.284,Z 337.978,A -85,B 0,C 180,E1 -5648.667,E2 -5648.667} C_VEL
LIN {X 0,Y 502.251,Z 342.09,A -85,B 0,C 180,E1 -5651.227,E2 -5651.227} C_VEL
LIN {X 0,Y 502.211,Z 347.669,A -85,B 0,C 180,E1 -5654.581,E2 -5654.581} C_VEL
LIN {X 0,Y 502.229,Z 349.706,A -85,B 0,C 180,E1 -5655.774,E2 -5655.774} C_VEL
LIN {X 0,Y 504.675,Z 362.824,A -85,B 0,C 180,E1 -5656.204,E2 -5656.204} C_VEL
LIN {X 0,Y 504.367,Z 375.662,A -85,B 0,C 180,E1 -5656.709,E2 -5656.709} C_VEL
LIN {X 0,Y 504.04,Z 387.264,A -85,B 0,C 180,E1 -5657.328,E2 -5657.328} C_VEL
LIN {X 0,Y 503.756,Z 398.72,A -85,B 0,C 180,E1 -5658.125,E2 -5658.125} C_VEL
LIN {X 0,Y 503.391,Z 409.188,A -85,B 0,C 180,E1 -5659.035,E2 -5659.035} C_VEL
LIN {X 0,Y 503.078,Z 417.741,A -85,B 0,C 180,E1 -5659.944,E2 -5659.944} C_VEL
LIN {X 0,Y 502.817,Z 425.617,A -85,B 0,C 180,E1 -5660.954,E2 -5660.954} C_VEL
LIN {X 0,Y 502.528,Z 433.319,A -85,B 0,C 180,E1 -5662.163,E2 -5662.163} C_VEL
LIN {X 0,Y 502.324,Z 440.382,A -85,B 0,C 180,E1 -5663.574,E2 -5663.574} C_VEL
LIN {X 0,Y 502.186,Z 445.089,A -85,B 0,C 180,E1 -5664.781,E2 -5664.781} C_VEL
LIN {X 0,Y 502.236,Z 448.689,A -85,B 0,C 180,E1 -5665.988,E2 -5665.988} C_VEL
LIN {X 0,Y 502.124,Z 450.555,A -85,B 0,C 180,E1 -5666.791,E2 -5666.791} C_VEL
LIN {X 0,Y 502.121,Z 451.96,A -85,B 0,C 180,E1 -5667.594,E2 -5667.594} C_VEL
LIN {X 0,Y 501.991,Z 453.578,A -85,B 0,C 180,E1 -5669.198,E2 -5669.198} C_VEL
LIN {X 0,Y 501.98,Z 453.814,A -85,B 0,C 180,E1 -5670,E2 -5670} C_VEL
LIN {X 0,Y 501.991,Z 453.63,A -85,B 0,C 180,E1 -5670.803,E2 -5670.803} C_VEL
LIN {X 0,Y 502.121,Z 452.081,A -85,B 0,C 180,E1 -5672.407,E2 -5672.407} C_VEL
LIN {X 0,Y 502.125,Z 450.728,A -85,B 0,C 180,E1 -5673.21,E2 -5673.21} C_VEL
LIN {X 0,Y 502.209,Z 447.867,A -85,B 0,C 180,E1 -5674.415,E2 -5674.415} C_VEL
LIN {X 0,Y 502.291,Z 443.987,A -85,B 0,C 180,E1 -5675.621,E2 -5675.621} C_VEL
LIN {X 0,Y 502.351,Z 438.985,A -85,B 0,C 180,E1 -5676.829,E2 -5676.829} C_VEL
LIN {X 0,Y 502.563,Z 432.682,A -85,B 0,C 180,E1 -5678.039,E2 -5678.039} C_VEL
LIN {X 0,Y 502.784,Z 424.792,A -85,B 0,C 180,E1 -5679.251,E2 -5679.251} C_VEL
LIN {X 0,Y 503.106,Z 416.747,A -85,B 0,C 180,E1 -5680.26,E2 -5680.26} C_VEL
LIN {X 0,Y 503.452,Z 406.929,A -85,B 0,C 180,E1 -5681.27,E2 -5681.27} C_VEL
LIN {X 0,Y 503.758,Z 397.271,A -85,B 0,C 180,E1 -5682.08,E2 -5682.08} C_VEL
LIN {X 0,Y 504.056,Z 386.431,A -85,B 0,C 180,E1 -5682.811,E2 -5682.811} C_VEL
LIN {X 0,Y 504.419,Z 374.251,A -85,B 0,C 180,E1 -5683.445,E2 -5683.445} C_VEL
LIN {X 0,Y 504.552,Z 362.059,A -85,B 0,C 180,E1 -5683.916,E2 -5683.916} C_VEL
LIN {X 0,Y 502.239,Z 349.681,A -85,B 0,C 180,E1 -5684.33,E2 -5684.33} C_VEL
LIN {X 0,Y 502.233,Z 343.637,A -85,B 0,C 180,E1 -5687.93,E2 -5687.93} C_VEL
LIN {X 0,Y 502.29,Z 339.479,A -85,B 0,C 180,E1 -5690.475,E2 -5690.475} C_VEL
LIN {X 0,Y 502.365,Z 335.408,A -85,B 0,C 180,E1 -5693.061,E2 -5693.061} C_VEL
LIN {X 0,Y 502.423,Z 331.328,A -85,B 0,C 180,E1 -5695.698,E2 -5695.698} C_VEL
LIN {X 0,Y 502.515,Z 327.219,A -85,B 0,C 180,E1 -5698.392,E2 -5698.392} C_VEL
LIN {X 0,Y 502.622,Z 322.638,A -85,B 0,C 180,E1 -5701.466,E2 -5701.466} C_VEL
LIN {X 0,Y 502.761,Z 318.288,A -85,B 0,C 180,E1 -5704.436,E2 -5704.436} C_VEL
LIN {X 0,Y 502.738,Z 317.531,A -85,B 0,C 180,E1 -5704.97,E2 -5704.97} C_VEL
LIN {X 0,Y 502.743,Z 316.86,A -85,B 0,C 180,E1 -5705.953,E2 -5705.953} C_VEL
LIN {X 0,Y 502.8,Z 316.856,A -85,B 0,C 180,E1 -5708.976,E2 -5708.976} C_VEL
LIN {X 0,Y 502.796,Z 316.856,A -85,B 0,C 180,E1 -5712.139,E2 -5712.139} C_VEL
LIN {X 0,Y 502.784,Z 316.859,A -85,B 0,C 180,E1 -5715.47,E2 -5715.47} C_VEL
LIN {X 0,Y 502.761,Z 316.861,A -85,B 0,C 180,E1 -5718.928,E2 -5718.928} C_VEL
LIN {X 0,Y 502.79,Z 316.857,A -85,B 0,C 180,E1 -5722.046,E2 -5722.046} C_VEL
LIN {X 0,Y 502.806,Z 316.852,A -85,B 0,C 180,E1 -5725.034,E2 -5725.034} C_VEL
LIN {X 0,Y 502.781,Z 316.855,A -85,B 0,C 180,E1 -5727.915,E2 -5727.915} C_VEL
LIN {X 0,Y 502.799,Z 316.854,A -85,B 0,C 180,E1 -5730.71,E2 -5730.71} C_VEL
LIN {X 0,Y 502.779,Z 316.856,A -85,B 0,C 180,E1 -5733.457,E2 -5733.457} C_VEL
LIN {X 0,Y 502.764,Z 316.86,A -85,B 0,C 180,E1 -5736.085,E2 -5736.085} C_VEL
LIN {X 0,Y 502.78,Z 316.856,A -85,B 0,C 180,E1 -5738.689,E2 -5738.689} C_VEL
LIN {X 0,Y 502.825,Z 316.853,A -85,B 0,C 180,E1 -5741.248,E2 -5741.248} C_VEL
LIN {X 0,Y 502.814,Z 316.849,A -85,B 0,C 180,E1 -5743.767,E2 -5743.767} C_VEL
LIN {X 0,Y 502.812,Z 316.854,A -85,B 0,C 180,E1 -5746.254,E2 -5746.254} C_VEL
LIN {X 0,Y 502.871,Z 316.845,A -85,B 0,C 180,E1 -5748.717,E2 -5748.717} C_VEL
LIN {X 0,Y 502.897,Z 316.843,A -85,B 0,C 180,E1 -5751.967,E2 -5751.967} C_VEL
LIN {X 0,Y 502.938,Z 316.837,A -85,B 0,C 180,E1 -5754.386,E2 -5754.386} C_VEL
LIN {X 0,Y 503.019,Z 316.824,A -85,B 0,C 180,E1 -5757.598,E2 -5757.598} C_VEL
LIN {X 0,Y 503.02,Z 316.829,A -85,B 0,C 180,E1 -5760,E2 -5760} C_VEL
LIN {X 0,Y 503.018,Z 316.826,A -85,B 0,C 180,E1 -5762.402,E2 -5762.402} C_VEL
LIN {X 0,Y 502.937,Z 316.838,A -85,B 0,C 180,E1 -5765.613,E2 -5765.613} C_VEL
LIN {X 0,Y 502.898,Z 316.842,A -85,B 0,C 180,E1 -5768.033,E2 -5768.033} C_VEL
LIN {X 0,Y 502.872,Z 316.842,A -85,B 0,C 180,E1 -5771.283,E2 -5771.283} C_VEL
LIN {X 0,Y 502.819,Z 316.85,A -85,B 0,C 180,E1 -5774.572,E2 -5774.572} C_VEL
LIN {X 0,Y 502.85,Z 316.847,A -85,B 0,C 180,E1 -5777.907,E2 -5777.907} C_VEL
LIN {X 0,Y 502.824,Z 316.853,A -85,B 0,C 180,E1 -5780.536,E2 -5780.536} C_VEL
LIN {X 0,Y 502.791,Z 316.854,A -85,B 0,C 180,E1 -5783.041,E2 -5783.041} C_VEL
LIN {X 0,Y 502.789,Z 316.859,A -85,B 0,C 180,E1 -5785.678,E2 -5785.678} C_VEL
LIN {X 0,Y 502.768,Z 316.856,A -85,B 0,C 180,E1 -5788.377,E2 -5788.377} C_VEL
LIN {X 0,Y 502.789,Z 316.858,A -85,B 0,C 180,E1 -5791.144,E2 -5791.144} C_VEL
LIN {X 0,Y 502.804,Z 316.856,A -85,B 0,C 180,E1 -5793.994,E2 -5793.994} C_VEL
LIN {X 0,Y 502.778,Z 316.857,A -85,B 0,C 180,E1 -5797.179,E2 -5797.179} C_VEL
LIN {X 0,Y 502.769,Z 316.855,A -85,B 0,C 180,E1 -5800.017,E2 -5800.017} C_VEL
LIN {X 0,Y 502.745,Z 316.862,A -85,B 0,C 180,E1 -5803.234,E2 -5803.234} C_VEL
LIN {X 0,Y 502.777,Z 316.857,A -85,B 0,C 180,E1 -5805.66,E2 -5805.66} C_VEL
LIN {X 0,Y 502.818,Z 316.852,A -85,B 0,C 180,E1 -5809.005,E2 -5809.005} C_VEL
LIN {X 0,Y 502.841,Z 316.992,A -85,B 0,C 180,E1 -5811.918,E2 -5811.918} C_VEL
LIN {X 0,Y 503.522,Z 321.76,A -85,B 0,C 180,E1 -5814.111,E2 -5814.111} C_VEL
LIN {X 0,Y 503.535,Z 326.308,A -85,B 0,C 180,E1 -5816.063,E2 -5816.063} C_VEL
LIN {X 0,Y 503.307,Z 333.114,A -85,B 0,C 180,E1 -5818.892,E2 -5818.892} C_VEL
LIN {X 0,Y 503.146,Z 339.901,A -85,B 0,C 180,E1 -5821.646,E2 -5821.646} C_VEL
LIN {X 0,Y 502.965,Z 347.813,A -85,B 0,C 180,E1 -5824.775,E2 -5824.775} C_VEL
LIN {X 0,Y 502.778,Z 355.692,A -85,B 0,C 180,E1 -5827.826,E2 -5827.826} C_VEL
LIN {X 0,Y 502.594,Z 363.483,A -85,B 0,C 180,E1 -5830.816,E2 -5830.816} C_VEL
LIN {X 0,Y 502.447,Z 371.274,A -85,B 0,C 180,E1 -5833.755,E2 -5833.755} C_VEL
LIN {X 0,Y 502.369,Z 376.491,A -85,B 0,C 180,E1 -5835.7,E2 -5835.7} C_VEL
LIN {X 0,Y 504.626,Z 389.927,A -85,B 0,C 180,E1 -5836.099,E2 -5836.099} C_VEL
LIN {X 0,Y 504.377,Z 403.239,A -85,B 0,C 180,E1 -5836.605,E2 -5836.605} C_VEL
LIN {X 0,Y 504.011,Z 415.861,A -85,B 0,C 180,E1 -5837.265,E2 -5837.265} C_VEL
LIN {X 0,Y 503.669,Z 426.904,A -85,B 0,C 180,E1 -5838.02,E2 -5838.02} C_VEL
LIN {X 0,Y 503.32,Z 437.537,A -85,B 0,C 180,E1 -5838.931,E2 -5838.931} C_VEL
LIN {X 0,Y 502.971,Z 447.112,A -85,B 0,C 180,E1 -5839.941,E2 -5839.941} C_VEL
LIN {X 0,Y 502.704,Z 454.959,A -85,B 0,C 180,E1 -5840.951,E2 -5840.951} C_VEL
LIN {X 0,Y 502.47,Z 462.62,A -85,B 0,C 180,E1 -5842.162,E2 -5842.162} C_VEL
LIN {X 0,Y 502.275,Z 469.679,A -85,B 0,C 180,E1 -5843.573,E2 -5843.573} C_VEL
LIN {X 0,Y 502.186,Z 474.372,A -85,B 0,C 180,E1 -5844.781,E2 -5844.781} C_VEL
LIN {X 0,Y 502.152,Z 477.957,A -85,B 0,C 180,E1 -5845.987,E2 -5845.987} C_VEL
LIN {X 0,Y 502.121,Z 479.807,A -85,B 0,C 180,E1 -5846.79,E2 -5846.79} C_VEL
LIN {X 0,Y 502.066,Z 481.195,A -85,B 0,C 180,E1 -5847.593,E2 -5847.593} C_VEL
LIN {X 0,Y 501.99,Z 482.786,A -85,B 0,C 180,E1 -5849.197,E2 -5849.197} C_VEL
LIN {X 0,Y 501.98,Z 483,A -85,B 0,C 180,E1 -5850,E2 -5850} C_VEL
LIN {X 0,Y 502.036,Z 482.185,A -85,B 0,C 180,E1 -5851.604,E2 -5851.604} C_VEL
LIN {X 0,Y 502.066,Z 481.198,A -85,B 0,C 180,E1 -5852.406,E2 -5852.406} C_VEL
LIN {X 0,Y 502.121,Z 479.811,A -85,B 0,C 180,E1 -5853.209,E2 -5853.209} C_VEL
LIN {X 0,Y 502.128,Z 476.897,A -85,B 0,C 180,E1 -5854.415,E2 -5854.415} C_VEL
LIN {X 0,Y 502.26,Z 472.95,A -85,B 0,C 180,E1 -5855.621,E2 -5855.621} C_VEL
LIN {X 0,Y 502.335,Z 466.979,A -85,B 0,C 180,E1 -5857.011,E2 -5857.011} C_VEL
LIN {X 0,Y 502.542,Z 460.239,A -85,B 0,C 180,E1 -5858.241,E2 -5858.241} C_VEL
LIN {X 0,Y 502.811,Z 451.995,A -85,B 0,C 180,E1 -5859.452,E2 -5859.452} C_VEL
LIN {X 0,Y 503.063,Z 443.544,A -85,B 0,C 180,E1 -5860.463,E2 -5860.463} C_VEL
LIN {X 0,Y 503.513,Z 433.101,A -85,B 0,C 180,E1 -5861.472,E2 -5861.472} C_VEL
LIN {X 0,Y 503.792,Z 421.437,A -85,B 0,C 180,E1 -5862.377,E2 -5862.377} C_VEL
LIN {X 0,Y 504.168,Z 409.501,A -85,B 0,C 180,E1 -5863.092,E2 -5863.092} C_VEL
LIN {X 0,Y 504.495,Z 397.183,A -85,B 0,C 180,E1 -5863.647,E2 -5863.647} C_VEL
LIN {X 0,Y 504.484,Z 388.654,A -85,B 0,C 180,E1 -5863.943,E2 -5863.943} C_VEL
LIN {X 0,Y 502.368,Z 376.493,A -85,B 0,C 180,E1 -5864.3,E2 -5864.3} C_VEL
LIN {X 0,Y 502.468,Z 369.05,A -85,B 0,C 180,E1 -5867.08,E2 -5867.08} C_VEL
LIN {X 0,Y 502.661,Z 361.259,A -85,B 0,C 180,E1 -5870.031,E2 -5870.031} C_VEL
LIN {X 0,Y 502.836,Z 353.467,A -85,B 0,C 180,E1 -5873.038,E2 -5873.038} C_VEL
LIN {X 0,Y 502.972,Z 345.541,A -85,B 0,C 180,E1 -5876.112,E2 -5876.112} C_VEL
LIN {X 0,Y 503.152,Z 338.741,A -85,B 0,C 180,E1 -5878.808,E2 -5878.808} C_VEL
LIN {X 0,Y 503.379,Z 331.829,A -85,B 0,C 180,E1 -5881.607,E2 -5881.607} C_VEL
LIN {X 0,Y 503.623,Z 324.029,A -85,B 0,C 180,E1 -5884.899,E2 -5884.899} C_VEL
LIN {X 0,Y 503.265,Z 319.516,A -85,B 0,C 180,E1 -5886.903,E2 -5886.903} C_VEL
LIN {X 0,Y 502.821,Z 316.855,A -85,B 0,C 180,E1 -5888.217,E2 -5888.217} C_VEL
LIN {X 0,Y 502.823,Z 316.853,A -85,B 0,C 180,E1 -5891.064,E2 -5891.064} C_VEL
LIN {X 0,Y 502.777,Z 316.861,A -85,B 0,C 180,E1 -5893.375,E2 -5893.375} C_VEL
LIN {X 0,Y 502.784,Z 316.858,A -85,B 0,C 180,E1 -5895.66,E2 -5895.66} C_VEL
LIN {X 0,Y 502.767,Z 316.861,A -85,B 0,C 180,E1 -5898.929,E2 -5898.929} C_VEL
LIN {X 0,Y 502.786,Z 316.856,A -85,B 0,C 180,E1 -5902.045,E2 -5902.045} C_VEL
LIN {X 0,Y 502.802,Z 316.853,A -85,B 0,C 180,E1 -5905.034,E2 -5905.034} C_VEL
LIN {X 0,Y 502.776,Z 316.858,A -85,B 0,C 180,E1 -5907.915,E2 -5907.915} C_VEL
LIN {X 0,Y 502.794,Z 316.858,A -85,B 0,C 180,E1 -5910.71,E2 -5910.71} C_VEL
LIN {X 0,Y 502.834,Z 316.846,A -85,B 0,C 180,E1 -5913.443,E2 -5913.443} C_VEL
LIN {X 0,Y 502.771,Z 316.861,A -85,B 0,C 180,E1 -5916.085,E2 -5916.085} C_VEL
LIN {X 0,Y 502.774,Z 316.856,A -85,B 0,C 180,E1 -5918.688,E2 -5918.688} C_VEL
LIN {X 0,Y 502.821,Z 316.853,A -85,B 0,C 180,E1 -5921.248,E2 -5921.248} C_VEL
LIN {X 0,Y 502.807,Z 316.852,A -85,B 0,C 180,E1 -5923.767,E2 -5923.767} C_VEL
LIN {X 0,Y 502.809,Z 316.856,A -85,B 0,C 180,E1 -5926.254,E2 -5926.254} C_VEL
LIN {X 0,Y 502.866,Z 316.843,A -85,B 0,C 180,E1 -5928.717,E2 -5928.717} C_VEL
LIN {X 0,Y 502.892,Z 316.843,A -85,B 0,C 180,E1 -5931.967,E2 -5931.967} C_VEL
LIN {X 0,Y 502.953,Z 316.836,A -85,B 0,C 180,E1 -5934.387,E2 -5934.387} C_VEL
LIN {X 0,Y 503.014,Z 316.827,A -85,B 0,C 180,E1 -5937.598,E2 -5937.598} C_VEL
LIN {X 0,Y 502.957,Z 316.832,A -85,B 0,C 180,E1 -5940.801,E2 -5940.801} C_VEL
LIN {X 0,Y 503.014,Z 316.824,A -85,B 0,C 180,E1 -5942.402,E2 -5942.402} C_VEL
LIN {X 0,Y 502.941,Z 316.837,A -85,B 0,C 180,E1 -5945.614,E2 -5945.614} C_VEL
LIN {X 0,Y 502.892,Z 316.843,A -85,B 0,C 180,E1 -5948.034,E2 -5948.034} C_VEL
LIN {X 0,Y 502.866,Z 316.845,A -85,B 0,C 180,E1 -5951.284,E2 -5951.284} C_VEL
LIN {X 0,Y 502.82,Z 316.849,A -85,B 0,C 180,E1 -5954.572,E2 -5954.572} C_VEL
LIN {X 0,Y 502.852,Z 316.845,A -85,B 0,C 180,E1 -5957.907,E2 -5957.907} C_VEL
LIN {X 0,Y 502.819,Z 316.853,A -85,B 0,C 180,E1 -5960.537,E2 -5960.537} C_VEL
LIN {X 0,Y 502.786,Z 316.855,A -85,B 0,C 180,E1 -5963.041,E2 -5963.041} C_VEL
LIN {X 0,Y 502.787,Z 316.857,A -85,B 0,C 180,E1 -5965.679,E2 -5965.679} C_VEL
LIN {X 0,Y 502.763,Z 316.857,A -85,B 0,C 180,E1 -5968.378,E2 -5968.378} C_VEL
LIN {X 0,Y 502.784,Z 316.856,A -85,B 0,C 180,E1 -5971.144,E2 -5971.144} C_VEL
LIN {X 0,Y 502.8,Z 316.854,A -85,B 0,C 180,E1 -5973.994,E2 -5973.994} C_VEL
LIN {X 0,Y 502.774,Z 316.858,A -85,B 0,C 180,E1 -5977.179,E2 -5977.179} C_VEL
LIN {X 0,Y 502.773,Z 316.857,A -85,B 0,C 180,E1 -5980.017,E2 -5980.017} C_VEL
LIN {X 0,Y 502.743,Z 316.86,A -85,B 0,C 180,E1 -5983.235,E2 -5983.235} C_VEL
LIN {X 0,Y 502.774,Z 316.855,A -85,B 0,C 180,E1 -5985.661,E2 -5985.661} C_VEL
LIN {X 0,Y 502.823,Z 316.85,A -85,B 0,C 180,E1 -5989.005,E2 -5989.005} C_VEL
LIN {X 0,Y 502.788,Z 316.855,A -85,B 0,C 180,E1 -5992.047,E2 -5992.047} C_VEL
LIN {X 0,Y 502.727,Z 316.863,A -85,B 0,C 180,E1 -5994.177,E2 -5994.177} C_VEL
LIN {X 0,Y 502.692,Z 317.393,A -85,B 0,C 180,E1 -5995.027,E2 -5995.027} C_VEL
LIN {X 0,Y 502.683,Z 320.528,A -85,B 0,C 180,E1 -5997.195,E2 -5997.195} C_VEL
LIN {X 0,Y 501.985,Z 321.571,A -85,B 0,C 180,E1 -5997.853,E2 -5997.853} C_VEL
LIN {X 0,Y 499.091,Z 323.467,A -85,B 0,C 180,E1 -5998.916,E2 -5998.916} C_VEL
LIN {X 0,Y 496.644,Z 325.006,A -85,B 0,C 180,E1 -5999.773,E2 -5999.773} C_VEL
LIN {X 0,Y 495.575,Z 326.105,A -85,B 0,C 180,E1 -6000.436,E2 -6000.436} C_VEL
LIN {X 0,Y 495.477,Z 326.447,A -85,B 0,C 180,E1 -6000.661,E2 -6000.661} C_VEL
LIN {X 0,Y 495.412,Z 330.457,A -85,B 0,C 180,E1 -6003.346,E2 -6003.346} C_VEL
LIN {X 0,Y 495.38,Z 334.041,A -85,B 0,C 180,E1 -6005.706,E2 -6005.706} C_VEL
LIN {X 0,Y 495.238,Z 338.128,A -85,B 0,C 180,E1 -6008.349,E2 -6008.349} C_VEL
LIN {X 0,Y 495.181,Z 342.245,A -85,B 0,C 180,E1 -6010.948,E2 -6010.948} C_VEL
LIN {X 0,Y 495.108,Z 346.416,A -85,B 0,C 180,E1 -6013.508,E2 -6013.508} C_VEL
LIN {X 0,Y 495.17,Z 349.861,A -85,B 0,C 180,E1 -6015.567,E2 -6015.567} C_VEL
LIN {X 0,Y 497.782,Z 363.819,A -85,B 0,C 180,E1 -6016.035,E2 -6016.035} C_VEL
LIN {X 0,Y 497.473,Z 375.891,A -85,B 0,C 180,E1 -6016.521,E2 -6016.521} C_VEL
LIN {X 0,Y 497.101,Z 387.768,A -85,B 0,C 180,E1 -6017.166,E2 -6017.166} C_VEL
LIN {X 0,Y 496.824,Z 398.943,A -85,B 0,C 180,E1 -6017.957,E2 -6017.957} C_VEL
LIN {X 0,Y 496.421,Z 409.411,A -85,B 0,C 180,E1 -6018.879,E2 -6018.879} C_VEL
LIN {X 0,Y 496.095,Z 417.962,A -85,B 0,C 180,E1 -6019.801,E2 -6019.801} C_VEL
LIN {X 0,Y 495.803,Z 425.837,A -85,B 0,C 180,E1 -6020.824,E2 -6020.824} C_VEL
LIN {X 0,Y 495.502,Z 433.538,A -85,B 0,C 180,E1 -6022.052,E2 -6022.052} C_VEL
LIN {X 0,Y 495.252,Z 440.6,A -85,B 0,C 180,E1 -6023.482,E2 -6023.482} C_VEL
LIN {X 0,Y 495.128,Z 445.306,A -85,B 0,C 180,E1 -6024.707,E2 -6024.707} C_VEL
LIN {X 0,Y 495.151,Z 448.907,A -85,B 0,C 180,E1 -6025.931,E2 -6025.931} C_VEL
LIN {X 0,Y 495.05,Z 450.771,A -85,B 0,C 180,E1 -6026.745,E2 -6026.745} C_VEL
LIN {X 0,Y 495.025,Z 452.176,A -85,B 0,C 180,E1 -6027.559,E2 -6027.559} C_VEL
LIN {X 0,Y 494.911,Z 453.793,A -85,B 0,C 180,E1 -6029.187,E2 -6029.187} C_VEL
LIN {X 0,Y 494.898,Z 454.03,A -85,B 0,C 180,E1 -6030,E2 -6030} C_VEL
LIN {X 0,Y 494.911,Z 453.845,A -85,B 0,C 180,E1 -6030.814,E2 -6030.814} C_VEL
LIN {X 0,Y 495.025,Z 452.295,A -85,B 0,C 180,E1 -6032.441,E2 -6032.441} C_VEL
LIN {X 0,Y 495.051,Z 450.942,A -85,B 0,C 180,E1 -6033.256,E2 -6033.256} C_VEL
LIN {X 0,Y 495.117,Z 448.081,A -85,B 0,C 180,E1 -6034.478,E2 -6034.478} C_VEL
LIN {X 0,Y 495.237,Z 444.2,A -85,B 0,C 180,E1 -6035.701,E2 -6035.701} C_VEL
LIN {X 0,Y 495.306,Z 439.197,A -85,B 0,C 180,E1 -6036.927,E2 -6036.927} C_VEL
LIN {X 0,Y 495.52,Z 432.894,A -85,B 0,C 180,E1 -6038.154,E2 -6038.154} C_VEL
LIN {X 0,Y 495.776,Z 425.003,A -85,B 0,C 180,E1 -6039.382,E2 -6039.382} C_VEL
LIN {X 0,Y 496.09,Z 416.958,A -85,B 0,C 180,E1 -6040.406,E2 -6040.406} C_VEL
LIN {X 0,Y 496.502,Z 407.137,A -85,B 0,C 180,E1 -6041.43,E2 -6041.43} C_VEL
LIN {X 0,Y 496.856,Z 396.218,A -85,B 0,C 180,E1 -6042.345,E2 -6042.345} C_VEL
LIN {X 0,Y 497.17,Z 385.278,A -85,B 0,C 180,E1 -6043.072,E2 -6043.072} C_VEL
LIN {X 0,Y 497.566,Z 373.325,A -85,B 0,C 180,E1 -6043.685,E2 -6043.685} C_VEL
LIN {X 0,Y 497.663,Z 363.016,A -85,B 0,C 180,E1 -6044.086,E2 -6044.086} C_VEL
LIN {X 0,Y 495.154,Z 349.835,A -85,B 0,C 180,E1 -6044.54,E2 -6044.54} C_VEL
LIN {X 0,Y 495.167,Z 343.792,A -85,B 0,C 180,E1 -6048.195,E2 -6048.195} C_VEL
LIN {X 0,Y 495.215,Z 339.629,A -85,B 0,C 180,E1 -6050.781,E2 -6050.781} C_VEL
LIN {X 0,Y 495.295,Z 335.549,A -85,B 0,C 180,E1 -6053.41,E2 -6053.41} C_VEL
LIN {X 0,Y 495.366,Z 331.454,A -85,B 0,C 180,E1 -6056.092,E2 -6056.092} C_VEL
LIN {X 0,Y 495.454,Z 327.335,A -85,B 0,C 180,E1 -6058.835,E2 -6058.835} C_VEL
LIN {X 0,Y 495.594,Z 323.129,A -85,B 0,C 180,E1 -6061.694,E2 -6061.694} C_VEL
LIN {X 0,Y 495.725,Z 318.82,A -85,B 0,C 180,E1 -6064.686,E2 -6064.686} C_VEL
LIN {X 0,Y 495.659,Z 317.745,A -85,B 0,C 180,E1 -6065.545,E2 -6065.545} C_VEL
LIN {X 0,Y 495.762,Z 317.734,A -85,B 0,C 180,E1 -6068.768,E2 -6068.768} C_VEL
LIN {X 0,Y 495.757,Z 317.733,A -85,B 0,C 180,E1 -6071.781,E2 -6071.781} C_VEL
LIN {X 0,Y 495.736,Z 317.733,A -85,B 0,C 180,E1 -6075.14,E2 -6075.14} C_VEL
LIN {X 0,Y 495.721,Z 317.734,A -85,B 0,C 180,E1 -6078.215,E2 -6078.215} C_VEL
LIN {X 0,Y 495.743,Z 317.733,A -85,B 0,C 180,E1 -6081.407,E2 -6081.407} C_VEL
LIN {X 0,Y 495.754,Z 317.733,A -85,B 0,C 180,E1 -6084.463,E2 -6084.463} C_VEL
LIN {X 0,Y 495.765,Z 317.734,A -85,B 0,C 180,E1 -6087.405,E2 -6087.405} C_VEL
LIN {X 0,Y 495.753,Z 317.729,A -85,B 0,C 180,E1 -6090.253,E2 -6090.253} C_VEL
LIN {X 0,Y 495.737,Z 317.733,A -85,B 0,C 180,E1 -6093.269,E2 -6093.269} C_VEL
LIN {X 0,Y 495.736,Z 317.735,A -85,B 0,C 180,E1 -6096.612,E2 -6096.612} C_VEL
LIN {X 0,Y 495.774,Z 317.732,A -85,B 0,C 180,E1 -6099.324,E2 -6099.324} C_VEL
LIN {X 0,Y 495.788,Z 317.726,A -85,B 0,C 180,E1 -6101.829,E2 -6101.829} C_VEL
LIN {X 0,Y 495.819,Z 317.726,A -85,B 0,C 180,E1 -6104.548,E2 -6104.548} C_VEL
LIN {X 0,Y 495.823,Z 317.724,A -85,B 0,C 180,E1 -6107.965,E2 -6107.965} C_VEL
LIN {X 0,Y 495.838,Z 317.722,A -85,B 0,C 180,E1 -6111.03,E2 -6111.03} C_VEL
LIN {X 0,Y 495.879,Z 317.716,A -85,B 0,C 180,E1 -6113.49,E2 -6113.49} C_VEL
LIN {X 0,Y 495.836,Z 317.723,A -85,B 0,C 180,E1 -6116.75,E2 -6116.75} C_VEL
LIN {X 0,Y 495.862,Z 317.722,A -85,B 0,C 180,E1 -6118.376,E2 -6118.376} C_VEL
LIN {X 0,Y 495.99,Z 317.704,A -85,B 0,C 180,E1 -6120,E2 -6120} C_VEL
LIN {X 0,Y 495.987,Z 317.702,A -85,B 0,C 180,E1 -6122.436,E2 -6122.436} C_VEL
LIN {X 0,Y 495.895,Z 317.715,A -85,B 0,C 180,E1 -6125.693,E2 -6125.693} C_VEL
LIN {X 0,Y 495.869,Z 317.718,A -85,B 0,C 180,E1 -6128.148,E2 -6128.148} C_VEL
LIN {X 0,Y 495.846,Z 317.718,A -85,B 0,C 180,E1 -6131.445,E2 -6131.445} C_VEL
LIN {X 0,Y 495.771,Z 317.728,A -85,B 0,C 180,E1 -6134.783,E2 -6134.783} C_VEL
LIN {X 0,Y 495.774,Z 317.732,A -85,B 0,C 180,E1 -6137.319,E2 -6137.319} C_VEL
LIN {X 0,Y 495.773,Z 317.729,A -85,B 0,C 180,E1 -6139.89,E2 -6139.89} C_VEL
LIN {X 0,Y 495.761,Z 317.73,A -85,B 0,C 180,E1 -6142.863,E2 -6142.863} C_VEL
LIN {X 0,Y 495.733,Z 317.734,A -85,B 0,C 180,E1 -6146.071,E2 -6146.071} C_VEL
LIN {X 0,Y 495.722,Z 317.735,A -85,B 0,C 180,E1 -6148.818,E2 -6148.818} C_VEL
LIN {X 0,Y 495.751,Z 317.731,A -85,B 0,C 180,E1 -6151.726,E2 -6151.726} C_VEL
LIN {X 0,Y 495.772,Z 317.731,A -85,B 0,C 180,E1 -6154.695,E2 -6154.695} C_VEL
LIN {X 0,Y 495.728,Z 317.738,A -85,B 0,C 180,E1 -6157.562,E2 -6157.562} C_VEL
LIN {X 0,Y 495.742,Z 317.731,A -85,B 0,C 180,E1 -6160.045,E2 -6160.045} C_VEL
LIN {X 0,Y 495.693,Z 317.742,A -85,B 0,C 180,E1 -6162.887,E2 -6162.887} C_VEL
LIN {X 0,Y 495.726,Z 317.737,A -85,B 0,C 180,E1 -6165.999,E2 -6165.999} C_VEL
LIN {X 0,Y 495.766,Z 317.732,A -85,B 0,C 180,E1 -6169.301,E2 -6169.301} C_VEL
LIN {X 0,Y 495.782,Z 317.772,A -85,B 0,C 180,E1 -6171.671,E2 -6171.671} C_VEL
LIN {X 0,Y 496.453,Z 322.291,A -85,B 0,C 180,E1 -6173.796,E2 -6173.796} C_VEL
LIN {X 0,Y 496.536,Z 327.322,A -85,B 0,C 180,E1 -6176.008,E2 -6176.008} C_VEL
LIN {X 0,Y 496.284,Z 334.127,A -85,B 0,C 180,E1 -6178.877,E2 -6178.877} C_VEL
LIN {X 0,Y 496.114,Z 342.043,A -85,B 0,C 180,E1 -6182.129,E2 -6182.129} C_VEL
LIN {X 0,Y 495.859,Z 349.504,A -85,B 0,C 180,E1 -6185.108,E2 -6185.108} C_VEL
LIN {X 0,Y 495.713,Z 356.798,A -85,B 0,C 180,E1 -6187.932,E2 -6187.932} C_VEL
LIN {X 0,Y 495.543,Z 364.596,A -85,B 0,C 180,E1 -6190.962,E2 -6190.962} C_VEL
LIN {X 0,Y 495.389,Z 373.5,A -85,B 0,C 180,E1 -6194.362,E2 -6194.362} C_VEL
LIN {X 0,Y 495.315,Z 376.491,A -85,B 0,C 180,E1 -6195.491,E2 -6195.491} C_VEL
LIN {X 0,Y 497.681,Z 390.309,A -85,B 0,C 180,E1 -6195.914,E2 -6195.914} C_VEL
LIN {X 0,Y 497.465,Z 403.238,A -85,B 0,C 180,E1 -6196.416,E2 -6196.416} C_VEL
LIN {X 0,Y 497.099,Z 414.672,A -85,B 0,C 180,E1 -6197.014,E2 -6197.014} C_VEL
LIN {X 0,Y 496.746,Z 425.587,A -85,B 0,C 180,E1 -6197.747,E2 -6197.747} C_VEL
LIN {X 0,Y 496.385,Z 436.467,A -85,B 0,C 180,E1 -6198.671,E2 -6198.671} C_VEL
LIN {X 0,Y 495.996,Z 445.332,A -85,B 0,C 180,E1 -6199.592,E2 -6199.592} C_VEL
LIN {X 0,Y 495.673,Z 454.959,A -85,B 0,C 180,E1 -6200.821,E2 -6200.821} C_VEL
LIN {X 0,Y 495.404,Z 462.621,A -85,B 0,C 180,E1 -6202.049,E2 -6202.049} C_VEL
LIN {X 0,Y 495.204,Z 469.678,A -85,B 0,C 180,E1 -6203.481,E2 -6203.481} C_VEL
LIN {X 0,Y 495.123,Z 474.372,A -85,B 0,C 180,E1 -6204.706,E2 -6204.706} C_VEL
LIN {X 0,Y 495.049,Z 477.958,A -85,B 0,C 180,E1 -6205.929,E2 -6205.929} C_VEL
LIN {X 0,Y 495.043,Z 479.807,A -85,B 0,C 180,E1 -6206.744,E2 -6206.744} C_VEL
LIN {X 0,Y 494.961,Z 482.183,A -85,B 0,C 180,E1 -6208.372,E2 -6208.372} C_VEL
LIN {X 0,Y 494.898,Z 483,A -85,B 0,C 180,E1 -6210,E2 -6210} C_VEL
LIN {X 0,Y 494.961,Z 482.185,A -85,B 0,C 180,E1 -6211.627,E2 -6211.627} C_VEL
LIN {X 0,Y 495.043,Z 479.811,A -85,B 0,C 180,E1 -6213.255,E2 -6213.255} C_VEL
LIN {X 0,Y 495.029,Z 476.897,A -85,B 0,C 180,E1 -6214.478,E2 -6214.478} C_VEL
LIN {X 0,Y 495.21,Z 471.804,A -85,B 0,C 180,E1 -6215.999,E2 -6215.999} C_VEL
LIN {X 0,Y 495.277,Z 465.871,A -85,B 0,C 180,E1 -6217.337,E2 -6217.337} C_VEL
LIN {X 0,Y 495.556,Z 459.006,A -85,B 0,C 180,E1 -6218.563,E2 -6218.563} C_VEL
LIN {X 0,Y 495.851,Z 450.417,A -85,B 0,C 180,E1 -6219.792,E2 -6219.792} C_VEL
LIN {X 0,Y 496.182,Z 441.604,A -85,B 0,C 180,E1 -6220.817,E2 -6220.817} C_VEL
LIN {X 0,Y 496.579,Z 430.751,A -85,B 0,C 180,E1 -6221.842,E2 -6221.842} C_VEL
LIN {X 0,Y 496.896,Z 420.221,A -85,B 0,C 180,E1 -6222.635,E2 -6222.635} C_VEL
LIN {X 0,Y 497.285,Z 407.512,A -85,B 0,C 180,E1 -6223.38,E2 -6223.38} C_VEL
LIN {X 0,Y 497.614,Z 395.882,A -85,B 0,C 180,E1 -6223.892,E2 -6223.892} C_VEL
LIN {X 0,Y 497.517,Z 389.084,A -85,B 0,C 180,E1 -6224.13,E2 -6224.13} C_VEL
LIN {X 0,Y 495.313,Z 376.493,A -85,B 0,C 180,E1 -6224.508,E2 -6224.508} C_VEL
LIN {X 0,Y 495.422,Z 369.05,A -85,B 0,C 180,E1 -6227.331,E2 -6227.331} C_VEL
LIN {X 0,Y 495.593,Z 362.372,A -85,B 0,C 180,E1 -6229.897,E2 -6229.897} C_VEL
LIN {X 0,Y 495.783,Z 354.715,A -85,B 0,C 180,E1 -6232.866,E2 -6232.866} C_VEL
LIN {X 0,Y 495.917,Z 346.551,A -85,B 0,C 180,E1 -6236.06,E2 -6236.06} C_VEL
LIN {X 0,Y 496.137,Z 339.771,A -85,B 0,C 180,E1 -6238.791,E2 -6238.791} C_VEL
LIN {X 0,Y 496.352,Z 332.952,A -85,B 0,C 180,E1 -6241.593,E2 -6241.593} C_VEL
LIN {X 0,Y 496.599,Z 325.374,A -85,B 0,C 180,E1 -6244.832,E2 -6244.832} C_VEL
LIN {X 0,Y 496.249,Z 320.583,A -85,B 0,C 180,E1 -6246.991,E2 -6246.991} C_VEL
LIN {X 0,Y 495.768,Z 317.734,A -85,B 0,C 180,E1 -6248.394,E2 -6248.394} C_VEL
LIN {X 0,Y 495.765,Z 317.732,A -85,B 0,C 180,E1 -6251.294,E2 -6251.294} C_VEL
LIN {X 0,Y 495.732,Z 317.738,A -85,B 0,C 180,E1 -6254,E2 -6254} C_VEL
LIN {X 0,Y 495.699,Z 317.742,A -85,B 0,C 180,E1 -6257.114,E2 -6257.114} C_VEL
LIN {X 0,Y 495.744,Z 317.73,A -85,B 0,C 180,E1 -6259.953,E2 -6259.953} C_VEL
LIN {X 0,Y 495.723,Z 317.738,A -85,B 0,C 180,E1 -6262.552,E2 -6262.552} C_VEL
LIN {X 0,Y 495.777,Z 317.73,A -85,B 0,C 180,E1 -6265.457,E2 -6265.457} C_VEL
LIN {X 0,Y 495.747,Z 317.732,A -85,B 0,C 180,E1 -6268.363,E2 -6268.363} C_VEL
LIN {X 0,Y 495.727,Z 317.733,A -85,B 0,C 180,E1 -6271.517,E2 -6271.517} C_VEL
LIN {X 0,Y 495.749,Z 317.731,A -85,B 0,C 180,E1 -6273.93,E2 -6273.93} C_VEL
LIN {X 0,Y 495.755,Z 317.731,A -85,B 0,C 180,E1 -6277.137,E2 -6277.137} C_VEL
LIN {X 0,Y 495.768,Z 317.73,A -85,B 0,C 180,E1 -6280.109,E2 -6280.109} C_VEL
LIN {X 0,Y 495.774,Z 317.732,A -85,B 0,C 180,E1 -6282.681,E2 -6282.681} C_VEL
LIN {X 0,Y 495.77,Z 317.728,A -85,B 0,C 180,E1 -6285.217,E2 -6285.217} C_VEL
LIN {X 0,Y 495.84,Z 317.719,A -85,B 0,C 180,E1 -6288.555,E2 -6288.555} C_VEL
LIN {X 0,Y 495.863,Z 317.719,A -85,B 0,C 180,E1 -6291.852,E2 -6291.852} C_VEL
LIN {X 0,Y 495.907,Z 317.713,A -85,B 0,C 180,E1 -6294.307,E2 -6294.307} C_VEL
LIN {X 0,Y 495.983,Z 317.703,A -85,B 0,C 180,E1 -6297.564,E2 -6297.564} C_VEL
LIN {X 0,Y 495.985,Z 317.705,A -85,B 0,C 180,E1 -6300,E2 -6300} C_VEL
LIN {X 0,Y 495.983,Z 317.7,A -85,B 0,C 180,E1 -6302.436,E2 -6302.436} C_VEL
LIN {X 0,Y 495.897,Z 317.714,A -85,B 0,C 180,E1 -6305.694,E2 -6305.694} C_VEL
LIN {X 0,Y 495.863,Z 317.719,A -85,B 0,C 180,E1 -6308.148,E2 -6308.148} C_VEL
LIN {X 0,Y 495.841,Z 317.721,A -85,B 0,C 180,E1 -6311.446,E2 -6311.446} C_VEL
LIN {X 0,Y 495.77,Z 317.728,A -85,B 0,C 180,E1 -6314.784,E2 -6314.784} C_VEL
LIN {X 0,Y 495.775,Z 317.731,A -85,B 0,C 180,E1 -6317.319,E2 -6317.319} C_VEL
LIN {X 0,Y 495.769,Z 317.729,A -85,B 0,C 180,E1 -6319.891,E2 -6319.891} C_VEL
LIN {X 0,Y 495.748,Z 317.733,A -85,B 0,C 180,E1 -6322.861,E2 -6322.861} C_VEL
LIN {X 0,Y 495.749,Z 317.733,A -85,B 0,C 180,E1 -6326.07,E2 -6326.07} C_VEL
LIN {X 0,Y 495.718,Z 317.737,A -85,B 0,C 180,E1 -6328.818,E2 -6328.818} C_VEL
LIN {X 0,Y 495.747,Z 317.73,A -85,B 0,C 180,E1 -6331.726,E2 -6331.726} C_VEL
LIN {X 0,Y 495.769,Z 317.731,A -85,B 0,C 180,E1 -6334.696,E2 -6334.696} C_VEL
LIN {X 0,Y 495.724,Z 317.737,A -85,B 0,C 180,E1 -6337.562,E2 -6337.562} C_VEL
LIN {X 0,Y 495.745,Z 317.733,A -85,B 0,C 180,E1 -6340.047,E2 -6340.047} C_VEL
LIN {X 0,Y 495.697,Z 317.741,A -85,B 0,C 180,E1 -6342.886,E2 -6342.886} C_VEL
LIN {X 0,Y 495.723,Z 317.735,A -85,B 0,C 180,E1 -6345.999,E2 -6345.999} C_VEL
LIN {X 0,Y 495.776,Z 317.729,A -85,B 0,C 180,E1 -6349.302,E2 -6349.302} C_VEL
LIN {X 0,Y 495.751,Z 317.733,A -85,B 0,C 180,E1 -6351.41,E2 -6351.41} C_VEL
LIN {X 0,Y 495.639,Z 317.748,A -85,B 0,C 180,E1 -6354.455,E2 -6354.455} C_VEL
LIN {X 0,Y 495.681,Z 320.272,A -85,B 0,C 180,E1 -6356.431,E2 -6356.431} C_VEL
LIN {X 0,Y 495.535,Z 324.44,A -85,B 0,C 180,E1 -6359.299,E2 -6359.299} C_VEL
LIN {X 0,Y 495.477,Z 326.447,A -85,B 0,C 180,E1 -6360.661,E2 -6360.661} C_VEL
LIN {X 0,Y 494.772,Z 327.513,A -85,B 0,C 180,E1 -6361.328,E2 -6361.328} C_VEL
LIN {X 0,Y 491.866,Z 329.433,A -85,B 0,C 180,E1 -6362.407,E2 -6362.407} C_VEL
LIN {X 0,Y 489.427,Z 330.987,A -85,B 0,C 180,E1 -6363.276,E2 -6363.276} C_VEL
LIN {X 0,Y 488.384,Z 332.105,A -85,B 0,C 180,E1 -6363.949,E2 -6363.949} C_VEL
LIN {X 0,Y 488.3,Z 332.451,A -85,B 0,C 180,E1 -6364.177,E2 -6364.177} C_VEL
LIN {X 0,Y 488.262,Z 335.55,A -85,B 0,C 180,E1 -6366.233,E2 -6366.233} C_VEL
LIN {X 0,Y 488.142,Z 340.361,A -85,B 0,C 180,E1 -6369.364,E2 -6369.364} C_VEL
LIN {X 0,Y 488.088,Z 345.194,A -85,B 0,C 180,E1 -6372.4,E2 -6372.4} C_VEL
LIN {X 0,Y 488.074,Z 350.052,A -85,B 0,C 180,E1 -6375.352,E2 -6375.352} C_VEL
LIN {X 0,Y 490.734,Z 363.678,A -85,B 0,C 180,E1 -6375.817,E2 -6375.817} C_VEL
LIN {X 0,Y 490.602,Z 376.12,A -85,B 0,C 180,E1 -6376.328,E2 -6376.328} C_VEL
LIN {X 0,Y 490.167,Z 388.239,A -85,B 0,C 180,E1 -6376.998,E2 -6376.998} C_VEL
LIN {X 0,Y 489.888,Z 399.166,A -85,B 0,C 180,E1 -6377.784,E2 -6377.784} C_VEL
LIN {X 0,Y 489.463,Z 409.633,A -85,B 0,C 180,E1 -6378.719,E2 -6378.719} C_VEL
LIN {X 0,Y 489.117,Z 418.183,A -85,B 0,C 180,E1 -6379.654,E2 -6379.654} C_VEL
LIN {X 0,Y 488.778,Z 426.058,A -85,B 0,C 180,E1 -6380.691,E2 -6380.691} C_VEL
LIN {X 0,Y 488.462,Z 433.757,A -85,B 0,C 180,E1 -6381.936,E2 -6381.936} C_VEL
LIN {X 0,Y 488.182,Z 440.819,A -85,B 0,C 180,E1 -6383.387,E2 -6383.387} C_VEL
LIN {X 0,Y 488.074,Z 445.523,A -85,B 0,C 180,E1 -6384.63,E2 -6384.63} C_VEL
LIN {X 0,Y 488.069,Z 449.124,A -85,B 0,C 180,E1 -6385.872,E2 -6385.872} C_VEL
LIN {X 0,Y 487.979,Z 450.988,A -85,B 0,C 180,E1 -6386.698,E2 -6386.698} C_VEL
LIN {X 0,Y 487.933,Z 452.393,A -85,B 0,C 180,E1 -6387.524,E2 -6387.524} C_VEL
LIN {X 0,Y 487.834,Z 454.008,A -85,B 0,C 180,E1 -6389.175,E2 -6389.175} C_VEL
LIN {X 0,Y 487.819,Z 454.244,A -85,B 0,C 180,E1 -6390,E2 -6390} C_VEL
LIN {X 0,Y 487.834,Z 454.059,A -85,B 0,C 180,E1 -6390.826,E2 -6390.826} C_VEL
LIN {X 0,Y 487.934,Z 452.51,A -85,B 0,C 180,E1 -6392.477,E2 -6392.477} C_VEL
LIN {X 0,Y 487.979,Z 451.156,A -85,B 0,C 180,E1 -6393.303,E2 -6393.303} C_VEL
LIN {X 0,Y 488.016,Z 448.296,A -85,B 0,C 180,E1 -6394.543,E2 -6394.543} C_VEL
LIN {X 0,Y 488.21,Z 443.351,A -85,B 0,C 180,E1 -6396.071,E2 -6396.071} C_VEL
LIN {X 0,Y 488.299,Z 437.439,A -85,B 0,C 180,E1 -6397.443,E2 -6397.443} C_VEL
LIN {X 0,Y 488.599,Z 430.658,A -85,B 0,C 180,E1 -6398.687,E2 -6398.687} C_VEL
LIN {X 0,Y 488.914,Z 422.193,A -85,B 0,C 180,E1 -6399.933,E2 -6399.933} C_VEL
LIN {X 0,Y 489.277,Z 413.483,A -85,B 0,C 180,E1 -6400.972,E2 -6400.972} C_VEL
LIN {X 0,Y 489.749,Z 402.752,A -85,B 0,C 180,E1 -6402.01,E2 -6402.01} C_VEL
LIN {X 0,Y 490.061,Z 391.256,A -85,B 0,C 180,E1 -6402.893,E2 -6402.893} C_VEL
LIN {X 0,Y 490.533,Z 379.918,A -85,B 0,C 180,E1 -6403.569,E2 -6403.569} C_VEL
LIN {X 0,Y 490.818,Z 367.274,A -85,B 0,C 180,E1 -6404.142,E2 -6404.142} C_VEL
LIN {X 0,Y 490.63,Z 363.217,A -85,B 0,C 180,E1 -6404.293,E2 -6404.293} C_VEL
LIN {X 0,Y 488.065,Z 350.024,A -85,B 0,C 180,E1 -6404.756,E2 -6404.756} C_VEL
LIN {X 0,Y 488.109,Z 343.959,A -85,B 0,C 180,E1 -6408.467,E2 -6408.467} C_VEL
LIN {X 0,Y 488.168,Z 339.785,A -85,B 0,C 180,E1 -6411.095,E2 -6411.095} C_VEL
LIN {X 0,Y 488.246,Z 335.701,A -85,B 0,C 180,E1 -6413.768,E2 -6413.768} C_VEL
LIN {X 0,Y 488.34,Z 331.084,A -85,B 0,C 180,E1 -6416.838,E2 -6416.838} C_VEL
LIN {X 0,Y 488.436,Z 327.453,A -85,B 0,C 180,E1 -6419.289,E2 -6419.289} C_VEL
LIN {X 0,Y 488.565,Z 323.294,A -85,B 0,C 180,E1 -6422.157,E2 -6422.157} C_VEL
LIN {X 0,Y 488.638,Z 319.101,A -85,B 0,C 180,E1 -6425.121,E2 -6425.121} C_VEL
LIN {X 0,Y 488.658,Z 318.617,A -85,B 0,C 180,E1 -6426.35,E2 -6426.35} C_VEL
LIN {X 0,Y 488.7,Z 318.611,A -85,B 0,C 180,E1 -6429.254,E2 -6429.254} C_VEL
LIN {X 0,Y 488.707,Z 318.61,A -85,B 0,C 180,E1 -6431.599,E2 -6431.599} C_VEL
LIN {X 0,Y 488.7,Z 318.608,A -85,B 0,C 180,E1 -6434.802,E2 -6434.802} C_VEL
LIN {X 0,Y 488.648,Z 318.619,A -85,B 0,C 180,E1 -6437.469,E2 -6437.469} C_VEL
LIN {X 0,Y 488.701,Z 318.61,A -85,B 0,C 180,E1 -6439.673,E2 -6439.673} C_VEL
LIN {X 0,Y 488.679,Z 318.614,A -85,B 0,C 180,E1 -6442.841,E2 -6442.841} C_VEL
LIN {X 0,Y 488.731,Z 318.607,A -85,B 0,C 180,E1 -6445.887,E2 -6445.887} C_VEL
LIN {X 0,Y 488.687,Z 318.611,A -85,B 0,C 180,E1 -6448.82,E2 -6448.82} C_VEL
LIN {X 0,Y 488.69,Z 318.61,A -85,B 0,C 180,E1 -6451.668,E2 -6451.668} C_VEL
LIN {X 0,Y 488.69,Z 318.613,A -85,B 0,C 180,E1 -6454.441,E2 -6454.441} C_VEL
LIN {X 0,Y 488.717,Z 318.608,A -85,B 0,C 180,E1 -6457.153,E2 -6457.153} C_VEL
LIN {X 0,Y 488.724,Z 318.607,A -85,B 0,C 180,E1 -6459.81,E2 -6459.81} C_VEL
LIN {X 0,Y 488.724,Z 318.606,A -85,B 0,C 180,E1 -6462.423,E2 -6462.423} C_VEL
LIN {X 0,Y 488.752,Z 318.604,A -85,B 0,C 180,E1 -6464.999,E2 -6464.999} C_VEL
LIN {X 0,Y 488.8,Z 318.6,A -85,B 0,C 180,E1 -6468.387,E2 -6468.387} C_VEL
LIN {X 0,Y 488.812,Z 318.597,A -85,B 0,C 180,E1 -6471.733,E2 -6471.733} C_VEL
LIN {X 0,Y 488.854,Z 318.591,A -85,B 0,C 180,E1 -6474.224,E2 -6474.224} C_VEL
LIN {X 0,Y 488.956,Z 318.575,A -85,B 0,C 180,E1 -6477.529,E2 -6477.529} C_VEL
LIN {X 0,Y 488.96,Z 318.58,A -85,B 0,C 180,E1 -6480,E2 -6480} C_VEL
LIN {X 0,Y 488.955,Z 318.578,A -85,B 0,C 180,E1 -6482.471,E2 -6482.471} C_VEL
LIN {X 0,Y 488.854,Z 318.592,A -85,B 0,C 180,E1 -6485.776,E2 -6485.776} C_VEL
LIN {X 0,Y 488.814,Z 318.598,A -85,B 0,C 180,E1 -6488.266,E2 -6488.266} C_VEL
LIN {X 0,Y 488.8,Z 318.597,A -85,B 0,C 180,E1 -6491.613,E2 -6491.613} C_VEL
LIN {X 0,Y 488.748,Z 318.604,A -85,B 0,C 180,E1 -6495.001,E2 -6495.001} C_VEL
LIN {X 0,Y 488.751,Z 318.605,A -85,B 0,C 180,E1 -6498.442,E2 -6498.442} C_VEL
LIN {X 0,Y 488.703,Z 318.611,A -85,B 0,C 180,E1 -6501.071,E2 -6501.071} C_VEL
LIN {X 0,Y 488.676,Z 318.615,A -85,B 0,C 180,E1 -6503.746,E2 -6503.746} C_VEL
LIN {X 0,Y 488.696,Z 318.608,A -85,B 0,C 180,E1 -6506.476,E2 -6506.476} C_VEL
LIN {X 0,Y 488.696,Z 318.614,A -85,B 0,C 180,E1 -6509.272,E2 -6509.272} C_VEL
LIN {X 0,Y 488.7,Z 318.612,A -85,B 0,C 180,E1 -6512.147,E2 -6512.147} C_VEL
LIN {X 0,Y 488.719,Z 318.608,A -85,B 0,C 180,E1 -6515.115,E2 -6515.115} C_VEL
LIN {X 0,Y 488.676,Z 318.612,A -85,B 0,C 180,E1 -6518.201,E2 -6518.201} C_VEL
LIN {X 0,Y 488.69,Z 318.608,A -85,B 0,C 180,E1 -6520.341,E2 -6520.341} C_VEL
LIN {X 0,Y 488.671,Z 318.613,A -85,B 0,C 180,E1 -6523.656,E2 -6523.656} C_VEL
LIN {X 0,Y 488.683,Z 318.616,A -85,B 0,C 180,E1 -6526.346,E2 -6526.346} C_VEL
LIN {X 0,Y 488.732,Z 318.61,A -85,B 0,C 180,E1 -6529.677,E2 -6529.677} C_VEL
LIN {X 0,Y 488.761,Z 318.816,A -85,B 0,C 180,E1 -6531.545,E2 -6531.545} C_VEL
LIN {X 0,Y 489.493,Z 323.84,A -85,B 0,C 180,E1 -6533.938,E2 -6533.938} C_VEL
LIN {X 0,Y 489.54,Z 328.344,A -85,B 0,C 180,E1 -6535.952,E2 -6535.952} C_VEL
LIN {X 0,Y 489.268,Z 335.141,A -85,B 0,C 180,E1 -6538.861,E2 -6538.861} C_VEL
LIN {X 0,Y 489.074,Z 343.054,A -85,B 0,C 180,E1 -6542.159,E2 -6542.159} C_VEL
LIN {X 0,Y 488.795,Z 350.957,A -85,B 0,C 180,E1 -6545.357,E2 -6545.357} C_VEL
LIN {X 0,Y 488.651,Z 357.798,A -85,B 0,C 180,E1 -6548.041,E2 -6548.041} C_VEL
LIN {X 0,Y 488.488,Z 365.709,A -85,B 0,C 180,E1 -6551.112,E2 -6551.112} C_VEL
LIN {X 0,Y 488.318,Z 374.828,A -85,B 0,C 180,E1 -6554.641,E2 -6554.641} C_VEL
LIN {X 0,Y 488.244,Z 376.491,A -85,B 0,C 180,E1 -6555.277,E2 -6555.277} C_VEL
LIN {X 0,Y 490.639,Z 390.309,A -85,B 0,C 180,E1 -6555.708,E2 -6555.708} C_VEL
LIN {X 0,Y 490.723,Z 397.172,A -85,B 0,C 180,E1 -6555.961,E2 -6555.961} C_VEL
LIN {X 0,Y 490.314,Z 409.488,A -85,B 0,C 180,E1 -6556.531,E2 -6556.531} C_VEL
LIN {X 0,Y 489.942,Z 421.524,A -85,B 0,C 180,E1 -6557.274,E2 -6557.274} C_VEL
LIN {X 0,Y 489.518,Z 433.091,A -85,B 0,C 180,E1 -6558.195,E2 -6558.195} C_VEL
LIN {X 0,Y 489.073,Z 443.538,A -85,B 0,C 180,E1 -6559.233,E2 -6559.233} C_VEL
LIN {X 0,Y 488.765,Z 451.99,A -85,B 0,C 180,E1 -6560.273,E2 -6560.273} C_VEL
LIN {X 0,Y 488.454,Z 460.234,A -85,B 0,C 180,E1 -6561.519,E2 -6561.519} C_VEL
LIN {X 0,Y 488.186,Z 466.874,A -85,B 0,C 180,E1 -6562.763,E2 -6562.763} C_VEL
LIN {X 0,Y 488.104,Z 472.949,A -85,B 0,C 180,E1 -6564.215,E2 -6564.215} C_VEL
LIN {X 0,Y 487.938,Z 476.894,A -85,B 0,C 180,E1 -6565.456,E2 -6565.456} C_VEL
LIN {X 0,Y 487.967,Z 479.806,A -85,B 0,C 180,E1 -6566.697,E2 -6566.697} C_VEL
LIN {X 0,Y 487.889,Z 482.182,A -85,B 0,C 180,E1 -6568.349,E2 -6568.349} C_VEL
LIN {X 0,Y 487.819,Z 483,A -85,B 0,C 180,E1 -6570,E2 -6570} C_VEL
LIN {X 0,Y 487.889,Z 482.184,A -85,B 0,C 180,E1 -6571.651,E2 -6571.651} C_VEL
LIN {X 0,Y 487.966,Z 479.811,A -85,B 0,C 180,E1 -6573.302,E2 -6573.302} C_VEL
LIN {X 0,Y 487.938,Z 476.896,A -85,B 0,C 180,E1 -6574.543,E2 -6574.543} C_VEL
LIN {X 0,Y 488.105,Z 472.95,A -85,B 0,C 180,E1 -6575.784,E2 -6575.784} C_VEL
LIN {X 0,Y 488.19,Z 466.878,A -85,B 0,C 180,E1 -6577.236,E2 -6577.236} C_VEL
LIN {X 0,Y 488.453,Z 460.239,A -85,B 0,C 180,E1 -6578.48,E2 -6578.48} C_VEL
LIN {X 0,Y 488.764,Z 451.996,A -85,B 0,C 180,E1 -6579.726,E2 -6579.726} C_VEL
LIN {X 0,Y 489.076,Z 443.545,A -85,B 0,C 180,E1 -6580.766,E2 -6580.766} C_VEL
LIN {X 0,Y 489.566,Z 433.099,A -85,B 0,C 180,E1 -6581.804,E2 -6581.804} C_VEL
LIN {X 0,Y 489.892,Z 421.895,A -85,B 0,C 180,E1 -6582.7,E2 -6582.7} C_VEL
LIN {X 0,Y 490.287,Z 411.416,A -85,B 0,C 180,E1 -6583.364,E2 -6583.364} C_VEL
LIN {X 0,Y 490.668,Z 399.779,A -85,B 0,C 180,E1 -6583.934,E2 -6583.934} C_VEL
LIN {X 0,Y 490.635,Z 390.323,A -85,B 0,C 180,E1 -6584.292,E2 -6584.292} C_VEL
LIN {X 0,Y 488.243,Z 376.493,A -85,B 0,C 180,E1 -6584.723,E2 -6584.723} C_VEL
LIN {X 0,Y 488.385,Z 369.05,A -85,B 0,C 180,E1 -6587.589,E2 -6587.589} C_VEL
LIN {X 0,Y 488.54,Z 362.346,A -85,B 0,C 180,E1 -6590.197,E2 -6590.197} C_VEL
LIN {X 0,Y 488.736,Z 355.04,A -85,B 0,C 180,E1 -6593.027,E2 -6593.027} C_VEL
LIN {X 0,Y 488.891,Z 347.563,A -85,B 0,C 180,E1 -6596.004,E2 -6596.004} C_VEL
LIN {X 0,Y 489.105,Z 340.795,A -85,B 0,C 180,E1 -6598.775,E2 -6598.775} C_VEL
LIN {X 0,Y 489.335,Z 334.019,A -85,B 0,C 180,E1 -6601.602,E2 -6601.602} C_VEL
LIN {X 0,Y 489.558,Z 327.216,A -85,B 0,C 180,E1 -6604.544,E2 -6604.544} C_VEL
LIN {X 0,Y 489.438,Z 322.939,A -85,B 0,C 180,E1 -6606.474,E2 -6606.474} C_VEL
LIN {X 0,Y 488.725,Z 318.611,A -85,B 0,C 180,E1 -6608.589,E2 -6608.589} C_VEL
LIN {X 0,Y 488.725,Z 318.612,A -85,B 0,C 180,E1 -6611.602,E2 -6611.602} C_VEL
LIN {X 0,Y 488.697,Z 318.614,A -85,B 0,C 180,E1 -6614.023,E2 -6614.023} C_VEL
LIN {X 0,Y 488.659,Z 318.617,A -85,B 0,C 180,E1 -6617.178,E2 -6617.178} C_VEL
LIN {X 0,Y 488.696,Z 318.608,A -85,B 0,C 180,E1 -6619.673,E2 -6619.673} C_VEL
LIN {X 0,Y 488.675,Z 318.613,A -85,B 0,C 180,E1 -6622.841,E2 -6622.841} C_VEL
LIN {X 0,Y 488.727,Z 318.608,A -85,B 0,C 180,E1 -6625.887,E2 -6625.887} C_VEL
LIN {X 0,Y 488.681,Z 318.615,A -85,B 0,C 180,E1 -6628.819,E2 -6628.819} C_VEL
LIN {X 0,Y 488.686,Z 318.61,A -85,B 0,C 180,E1 -6631.667,E2 -6631.667} C_VEL
LIN {X 0,Y 488.704,Z 318.612,A -85,B 0,C 180,E1 -6634.442,E2 -6634.442} C_VEL
LIN {X 0,Y 488.718,Z 318.608,A -85,B 0,C 180,E1 -6637.153,E2 -6637.153} C_VEL
LIN {X 0,Y 488.719,Z 318.61,A -85,B 0,C 180,E1 -6639.81,E2 -6639.81} C_VEL
LIN {X 0,Y 488.722,Z 318.609,A -85,B 0,C 180,E1 -6642.423,E2 -6642.423} C_VEL
LIN {X 0,Y 488.745,Z 318.604,A -85,B 0,C 180,E1 -6644.999,E2 -6644.999} C_VEL
LIN {X 0,Y 488.794,Z 318.598,A -85,B 0,C 180,E1 -6648.387,E2 -6648.387} C_VEL
LIN {X 0,Y 488.808,Z 318.599,A -85,B 0,C 180,E1 -6651.733,E2 -6651.733} C_VEL
LIN {X 0,Y 488.863,Z 318.59,A -85,B 0,C 180,E1 -6654.224,E2 -6654.224} C_VEL
LIN {X 0,Y 488.951,Z 318.579,A -85,B 0,C 180,E1 -6657.529,E2 -6657.529} C_VEL
LIN {X 0,Y 488.956,Z 318.581,A -85,B 0,C 180,E1 -6660,E2 -6660} C_VEL
LIN {X 0,Y 488.951,Z 318.576,A -85,B 0,C 180,E1 -6662.471,E2 -6662.471} C_VEL
LIN {X 0,Y 488.855,Z 318.591,A -85,B 0,C 180,E1 -6665.776,E2 -6665.776} C_VEL
LIN {X 0,Y 488.808,Z 318.598,A -85,B 0,C 180,E1 -6668.267,E2 -6668.267} C_VEL
LIN {X 0,Y 488.795,Z 318.6,A -85,B 0,C 180,E1 -6671.613,E2 -6671.613} C_VEL
LIN {X 0,Y 488.745,Z 318.604,A -85,B 0,C 180,E1 -6675.001,E2 -6675.001} C_VEL
LIN {X 0,Y 488.745,Z 318.604,A -85,B 0,C 180,E1 -6678.443,E2 -6678.443} C_VEL
LIN {X 0,Y 488.699,Z 318.611,A -85,B 0,C 180,E1 -6681.071,E2 -6681.071} C_VEL
LIN {X 0,Y 488.671,Z 318.616,A -85,B 0,C 180,E1 -6683.747,E2 -6683.747} C_VEL
LIN {X 0,Y 488.713,Z 318.609,A -85,B 0,C 180,E1 -6686.928,E2 -6686.928} C_VEL
LIN {X 0,Y 488.695,Z 318.609,A -85,B 0,C 180,E1 -6690.362,E2 -6690.362} C_VEL
LIN {X 0,Y 488.728,Z 318.605,A -85,B 0,C 180,E1 -6693.485,E2 -6693.485} C_VEL
LIN {X 0,Y 488.682,Z 318.615,A -85,B 0,C 180,E1 -6696.357,E2 -6696.357} C_VEL
LIN {X 0,Y 488.689,Z 318.614,A -85,B 0,C 180,E1 -6699.256,E2 -6699.256} C_VEL
LIN {X 0,Y 488.66,Z 318.617,A -85,B 0,C 180,E1 -6702.529,E2 -6702.529} C_VEL
LIN {X 0,Y 488.696,Z 318.608,A -85,B 0,C 180,E1 -6705.198,E2 -6705.198} C_VEL
LIN {X 0,Y 488.708,Z 318.61,A -85,B 0,C 180,E1 -6708.4,E2 -6708.4} C_VEL
LIN {X 0,Y 488.737,Z 318.607,A -85,B 0,C 180,E1 -6710.943,E2 -6710.943} C_VEL
LIN {X 0,Y 488.641,Z 318.618,A -85,B 0,C 180,E1 -6713.866,E2 -6713.866} C_VEL
LIN {X 0,Y 488.621,Z 319.233,A -85,B 0,C 180,E1 -6715.07,E2 -6715.07} C_VEL
LIN {X 0,Y 488.556,Z 323.486,A -85,B 0,C 180,E1 -6718.074,E2 -6718.074} C_VEL
LIN {X 0,Y 488.423,Z 328.281,A -85,B 0,C 180,E1 -6721.371,E2 -6721.371} C_VEL
LIN {X 0,Y 488.3,Z 332.451,A -85,B 0,C 180,E1 -6724.177,E2 -6724.177} C_VEL
LIN {X 0,Y 487.63,Z 333.535,A -85,B 0,C 180,E1 -6724.853,E2 -6724.853} C_VEL
LIN {X 0,Y 484.747,Z 335.474,A -85,B 0,C 180,E1 -6725.947,E2 -6725.947} C_VEL
LIN {X 0,Y 482.289,Z 337.043,A -85,B 0,C 180,E1 -6726.827,E2 -6726.827} C_VEL
LIN {X 0,Y 481.209,Z 338.174,A -85,B 0,C 180,E1 -6727.51,E2 -6727.51} C_VEL
LIN {X 0,Y 481.108,Z 338.533,A -85,B 0,C 180,E1 -6727.741,E2 -6727.741} C_VEL
LIN {X 0,Y 481.041,Z 342.577,A -85,B 0,C 180,E1 -6730.366,E2 -6730.366} C_VEL
LIN {X 0,Y 480.96,Z 346.774,A -85,B 0,C 180,E1 -6733.008,E2 -6733.008} C_VEL
LIN {X 0,Y 481.006,Z 350.252,A -85,B 0,C 180,E1 -6735.132,E2 -6735.132} C_VEL
LIN {X 0,Y 483.663,Z 363.536,A -85,B 0,C 180,E1 -6735.592,E2 -6735.592} C_VEL
LIN {X 0,Y 484.007,Z 366.556,A -85,B 0,C 180,E1 -6735.71,E2 -6735.71} C_VEL
LIN {X 0,Y 483.656,Z 378.462,A -85,B 0,C 180,E1 -6736.235,E2 -6736.235} C_VEL
LIN {X 0,Y 483.238,Z 390.179,A -85,B 0,C 180,E1 -6736.925,E2 -6736.925} C_VEL
LIN {X 0,Y 482.873,Z 401.957,A -85,B 0,C 180,E1 -6737.817,E2 -6737.817} C_VEL
LIN {X 0,Y 482.466,Z 410.915,A -85,B 0,C 180,E1 -6738.659,E2 -6738.659} C_VEL
LIN {X 0,Y 482.053,Z 420.101,A -85,B 0,C 180,E1 -6739.713,E2 -6739.713} C_VEL
LIN {X 0,Y 481.65,Z 429.017,A -85,B 0,C 180,E1 -6740.976,E2 -6740.976} C_VEL
LIN {X 0,Y 481.329,Z 436.195,A -85,B 0,C 180,E1 -6742.238,E2 -6742.238} C_VEL
LIN {X 0,Y 481.136,Z 442.438,A -85,B 0,C 180,E1 -6743.634,E2 -6743.634} C_VEL
LIN {X 0,Y 480.913,Z 447.058,A -85,B 0,C 180,E1 -6744.97,E2 -6744.97} C_VEL
LIN {X 0,Y 480.973,Z 449.341,A -85,B 0,C 180,E1 -6745.811,E2 -6745.811} C_VEL
LIN {X 0,Y 480.91,Z 451.204,A -85,B 0,C 180,E1 -6746.649,E2 -6746.649} C_VEL
LIN {X 0,Y 480.846,Z 452.609,A -85,B 0,C 180,E1 -6747.487,E2 -6747.487} C_VEL
LIN {X 0,Y 480.823,Z 453.606,A -85,B 0,C 180,E1 -6748.325,E2 -6748.325} C_VEL
LIN {X 0,Y 480.743,Z 454.459,A -85,B 0,C 180,E1 -6750,E2 -6750} C_VEL
LIN {X 0,Y 480.76,Z 454.273,A -85,B 0,C 180,E1 -6750.838,E2 -6750.838} C_VEL
LIN {X 0,Y 480.824,Z 453.689,A -85,B 0,C 180,E1 -6751.676,E2 -6751.676} C_VEL
LIN {X 0,Y 480.91,Z 451.37,A -85,B 0,C 180,E1 -6753.351,E2 -6753.351} C_VEL
LIN {X 0,Y 480.92,Z 448.51,A -85,B 0,C 180,E1 -6754.61,E2 -6754.61} C_VEL
LIN {X 0,Y 481.133,Z 444.626,A -85,B 0,C 180,E1 -6755.869,E2 -6755.869} C_VEL
LIN {X 0,Y 481.197,Z 439.621,A -85,B 0,C 180,E1 -6757.132,E2 -6757.132} C_VEL
LIN {X 0,Y 481.451,Z 433.318,A -85,B 0,C 180,E1 -6758.394,E2 -6758.394} C_VEL
LIN {X 0,Y 481.778,Z 425.425,A -85,B 0,C 180,E1 -6759.658,E2 -6759.658} C_VEL
LIN {X 0,Y 482.114,Z 417.378,A -85,B 0,C 180,E1 -6760.712,E2 -6760.712} C_VEL
LIN {X 0,Y 482.594,Z 407.555,A -85,B 0,C 180,E1 -6761.764,E2 -6761.764} C_VEL
LIN {X 0,Y 482.996,Z 396.584,A -85,B 0,C 180,E1 -6762.709,E2 -6762.709} C_VEL
LIN {X 0,Y 483.341,Z 385.689,A -85,B 0,C 180,E1 -6763.453,E2 -6763.453} C_VEL
LIN {X 0,Y 483.801,Z 373.729,A -85,B 0,C 180,E1 -6764.083,E2 -6764.083} C_VEL
LIN {X 0,Y 483.878,Z 364.934,A -85,B 0,C 180,E1 -6764.443,E2 -6764.443} C_VEL
LIN {X 0,Y 481.471,Z 352.638,A -85,B 0,C 180,E1 -6764.884,E2 -6764.884} C_VEL
LIN {X 0,Y 481.015,Z 350.221,A -85,B 0,C 180,E1 -6764.977,E2 -6764.977} C_VEL
LIN {X 0,Y 481.046,Z 344.13,A -85,B 0,C 180,E1 -6768.749,E2 -6768.749} C_VEL
LIN {X 0,Y 481.088,Z 339.945,A -85,B 0,C 180,E1 -6771.421,E2 -6771.421} C_VEL
LIN {X 0,Y 481.2,Z 335.842,A -85,B 0,C 180,E1 -6774.138,E2 -6774.138} C_VEL
LIN {X 0,Y 481.281,Z 331.56,A -85,B 0,C 180,E1 -6777.03,E2 -6777.03} C_VEL
LIN {X 0,Y 481.403,Z 327.573,A -85,B 0,C 180,E1 -6779.76,E2 -6779.76} C_VEL
LIN {X 0,Y 481.522,Z 323.402,A -85,B 0,C 180,E1 -6782.685,E2 -6782.685} C_VEL
LIN {X 0,Y 481.583,Z 319.9,A -85,B 0,C 180,E1 -6785.19,E2 -6785.19} C_VEL
LIN {X 0,Y 481.56,Z 319.5,A -85,B 0,C 180,E1 -6785.716,E2 -6785.716} C_VEL
LIN {X 0,Y 481.669,Z 319.489,A -85,B 0,C 180,E1 -6788.859,E2 -6788.859} C_VEL
LIN {X 0,Y 481.653,Z 319.492,A -85,B 0,C 180,E1 -6791.912,E2 -6791.912} C_VEL
LIN {X 0,Y 481.654,Z 319.485,A -85,B 0,C 180,E1 -6794.457,E2 -6794.457} C_VEL
LIN {X 0,Y 481.613,Z 319.492,A -85,B 0,C 180,E1 -6796.855,E2 -6796.855} C_VEL
LIN {X 0,Y 481.654,Z 319.488,A -85,B 0,C 180,E1 -6800.057,E2 -6800.057} C_VEL
LIN {X 0,Y 481.626,Z 319.491,A -85,B 0,C 180,E1 -6803.253,E2 -6803.253} C_VEL
LIN {X 0,Y 481.707,Z 319.481,A -85,B 0,C 180,E1 -6806.33,E2 -6806.33} C_VEL
LIN {X 0,Y 481.643,Z 319.491,A -85,B 0,C 180,E1 -6809.418,E2 -6809.418} C_VEL
LIN {X 0,Y 481.646,Z 319.488,A -85,B 0,C 180,E1 -6812.165,E2 -6812.165} C_VEL
LIN {X 0,Y 481.67,Z 319.486,A -85,B 0,C 180,E1 -6814.967,E2 -6814.967} C_VEL
LIN {X 0,Y 481.645,Z 319.49,A -85,B 0,C 180,E1 -6817.704,E2 -6817.704} C_VEL
LIN {X 0,Y 481.703,Z 319.481,A -85,B 0,C 180,E1 -6820.393,E2 -6820.393} C_VEL
LIN {X 0,Y 481.682,Z 319.486,A -85,B 0,C 180,E1 -6823.033,E2 -6823.033} C_VEL
LIN {X 0,Y 481.674,Z 319.484,A -85,B 0,C 180,E1 -6825.638,E2 -6825.638} C_VEL
LIN {X 0,Y 481.746,Z 319.479,A -85,B 0,C 180,E1 -6828.215,E2 -6828.215} C_VEL
LIN {X 0,Y 481.758,Z 319.476,A -85,B 0,C 180,E1 -6831.612,E2 -6831.612} C_VEL
LIN {X 0,Y 481.815,Z 319.467,A -85,B 0,C 180,E1 -6834.14,E2 -6834.14} C_VEL
LIN {X 0,Y 481.922,Z 319.452,A -85,B 0,C 180,E1 -6837.492,E2 -6837.492} C_VEL
LIN {X 0,Y 481.93,Z 319.455,A -85,B 0,C 180,E1 -6840,E2 -6840} C_VEL
LIN {X 0,Y 481.921,Z 319.454,A -85,B 0,C 180,E1 -6842.507,E2 -6842.507} C_VEL
LIN {X 0,Y 481.814,Z 319.468,A -85,B 0,C 180,E1 -6845.86,E2 -6845.86} C_VEL
LIN {X 0,Y 481.759,Z 319.478,A -85,B 0,C 180,E1 -6848.388,E2 -6848.388} C_VEL
LIN {X 0,Y 481.746,Z 319.477,A -85,B 0,C 180,E1 -6851.785,E2 -6851.785} C_VEL
LIN {X 0,Y 481.732,Z 319.478,A -85,B 0,C 180,E1 -6855.225,E2 -6855.225} C_VEL
LIN {X 0,Y 481.708,Z 319.482,A -85,B 0,C 180,E1 -6858.722,E2 -6858.722} C_VEL
LIN {X 0,Y 481.643,Z 319.489,A -85,B 0,C 180,E1 -6861.395,E2 -6861.395} C_VEL
LIN {X 0,Y 481.655,Z 319.489,A -85,B 0,C 180,E1 -6864.114,E2 -6864.114} C_VEL
LIN {X 0,Y 481.678,Z 319.484,A -85,B 0,C 180,E1 -6867.124,E2 -6867.124} C_VEL
LIN {X 0,Y 481.662,Z 319.487,A -85,B 0,C 180,E1 -6869.742,E2 -6869.742} C_VEL
LIN {X 0,Y 481.669,Z 319.487,A -85,B 0,C 180,E1 -6872.675,E2 -6872.675} C_VEL
LIN {X 0,Y 481.639,Z 319.493,A -85,B 0,C 180,E1 -6875.709,E2 -6875.709} C_VEL
LIN {X 0,Y 481.664,Z 319.486,A -85,B 0,C 180,E1 -6878.86,E2 -6878.86} C_VEL
LIN {X 0,Y 481.613,Z 319.491,A -85,B 0,C 180,E1 -6882.165,E2 -6882.165} C_VEL
LIN {X 0,Y 481.651,Z 319.491,A -85,B 0,C 180,E1 -6884.458,E2 -6884.458} C_VEL
LIN {X 0,Y 481.647,Z 319.492,A -85,B 0,C 180,E1 -6887.84,E2 -6887.84} C_VEL
LIN {X 0,Y 481.696,Z 319.487,A -85,B 0,C 180,E1 -6891.144,E2 -6891.144} C_VEL
LIN {X 0,Y 482.399,Z 323.761,A -85,B 0,C 180,E1 -6893.322,E2 -6893.322} C_VEL
LIN {X 0,Y 482.56,Z 328.253,A -85,B 0,C 180,E1 -6895.39,E2 -6895.39} C_VEL
LIN {X 0,Y 482.33,Z 335.022,A -85,B 0,C 180,E1 -6898.362,E2 -6898.362} C_VEL
LIN {X 0,Y 482.078,Z 341.808,A -85,B 0,C 180,E1 -6901.243,E2 -6901.243} C_VEL
LIN {X 0,Y 481.838,Z 348.571,A -85,B 0,C 180,E1 -6904.051,E2 -6904.051} C_VEL
LIN {X 0,Y 481.646,Z 356.535,A -85,B 0,C 180,E1 -6907.258,E2 -6907.258} C_VEL
LIN {X 0,Y 481.475,Z 364.482,A -85,B 0,C 180,E1 -6910.383,E2 -6910.383} C_VEL
LIN {X 0,Y 481.239,Z 373.5,A -85,B 0,C 180,E1 -6913.89,E2 -6913.89} C_VEL
LIN {X 0,Y 481.174,Z 376.491,A -85,B 0,C 180,E1 -6915.055,E2 -6915.055} C_VEL
LIN {X 0,Y 483.569,Z 390.309,A -85,B 0,C 180,E1 -6915.494,E2 -6915.494} C_VEL
LIN {X 0,Y 483.948,Z 394.499,A -85,B 0,C 180,E1 -6915.653,E2 -6915.653} C_VEL
LIN {X 0,Y 483.553,Z 406.508,A -85,B 0,C 180,E1 -6916.178,E2 -6916.178} C_VEL
LIN {X 0,Y 483.129,Z 418.18,A -85,B 0,C 180,E1 -6916.861,E2 -6916.861} C_VEL
LIN {X 0,Y 482.726,Z 429.483,A -85,B 0,C 180,E1 -6917.706,E2 -6917.706} C_VEL
LIN {X 0,Y 482.302,Z 439.644,A -85,B 0,C 180,E1 -6918.655,E2 -6918.655} C_VEL
LIN {X 0,Y 481.877,Z 448.784,A -85,B 0,C 180,E1 -6919.708,E2 -6919.708} C_VEL
LIN {X 0,Y 481.531,Z 457.686,A -85,B 0,C 180,E1 -6920.973,E2 -6920.973} C_VEL
LIN {X 0,Y 481.208,Z 464.847,A -85,B 0,C 180,E1 -6922.236,E2 -6922.236} C_VEL
LIN {X 0,Y 481.048,Z 470.356,A -85,B 0,C 180,E1 -6923.447,E2 -6923.447} C_VEL
LIN {X 0,Y 480.998,Z 474.372,A -85,B 0,C 180,E1 -6924.55,E2 -6924.55} C_VEL
LIN {X 0,Y 480.847,Z 477.957,A -85,B 0,C 180,E1 -6925.809,E2 -6925.809} C_VEL
LIN {X 0,Y 480.891,Z 479.806,A -85,B 0,C 180,E1 -6926.648,E2 -6926.648} C_VEL
LIN {X 0,Y 480.79,Z 482.182,A -85,B 0,C 180,E1 -6928.324,E2 -6928.324} C_VEL
LIN {X 0,Y 480.743,Z 483,A -85,B 0,C 180,E1 -6930,E2 -6930} C_VEL
LIN {X 0,Y 480.79,Z 482.184,A -85,B 0,C 180,E1 -6931.675,E2 -6931.675} C_VEL
LIN {X 0,Y 480.891,Z 479.811,A -85,B 0,C 180,E1 -6933.351,E2 -6933.351} C_VEL
LIN {X 0,Y 480.854,Z 476.896,A -85,B 0,C 180,E1 -6934.61,E2 -6934.61} C_VEL
LIN {X 0,Y 481.023,Z 472.95,A -85,B 0,C 180,E1 -6935.87,E2 -6935.87} C_VEL
LIN {X 0,Y 481.115,Z 466.878,A -85,B 0,C 180,E1 -6937.343,E2 -6937.343} C_VEL
LIN {X 0,Y 481.425,Z 460.239,A -85,B 0,C 180,E1 -6938.605,E2 -6938.605} C_VEL
LIN {X 0,Y 481.755,Z 451.996,A -85,B 0,C 180,E1 -6939.869,E2 -6939.869} C_VEL
LIN {X 0,Y 482.082,Z 443.545,A -85,B 0,C 180,E1 -6940.924,E2 -6940.924} C_VEL
LIN {X 0,Y 482.581,Z 433.098,A -85,B 0,C 180,E1 -6941.977,E2 -6941.977} C_VEL
LIN {X 0,Y 482.967,Z 421.886,A -85,B 0,C 180,E1 -6942.886,E2 -6942.886} C_VEL
LIN {X 0,Y 483.418,Z 409.498,A -85,B 0,C 180,E1 -6943.664,E2 -6943.664} C_VEL
LIN {X 0,Y 483.816,Z 397.18,A -85,B 0,C 180,E1 -6944.242,E2 -6944.242} C_VEL
LIN {X 0,Y 483.745,Z 391.464,A -85,B 0,C 180,E1 -6944.459,E2 -6944.459} C_VEL
LIN {X 0,Y 481.535,Z 378.441,A -85,B 0,C 180,E1 -6944.89,E2 -6944.89} C_VEL
LIN {X 0,Y 481.18,Z 376.424,A -85,B 0,C 180,E1 -6944.971,E2 -6944.971} C_VEL
LIN {X 0,Y 481.34,Z 367.698,A -85,B 0,C 180,E1 -6948.366,E2 -6948.366} C_VEL
LIN {X 0,Y 481.519,Z 361.149,A -85,B 0,C 180,E1 -6950.915,E2 -6950.915} C_VEL
LIN {X 0,Y 481.714,Z 353.063,A -85,B 0,C 180,E1 -6954.11,E2 -6954.11} C_VEL
LIN {X 0,Y 481.95,Z 345.574,A -85,B 0,C 180,E1 -6957.186,E2 -6957.186} C_VEL
LIN {X 0,Y 482.219,Z 338.413,A -85,B 0,C 180,E1 -6960.185,E2 -6960.185} C_VEL
LIN {X 0,Y 482.476,Z 330.503,A -85,B 0,C 180,E1 -6963.608,E2 -6963.608} C_VEL
LIN {X 0,Y 482.595,Z 326,A -85,B 0,C 180,E1 -6965.627,E2 -6965.627} C_VEL
LIN {X 0,Y 481.945,Z 320.921,A -85,B 0,C 180,E1 -6968.051,E2 -6968.051} C_VEL
LIN {X 0,Y 481.714,Z 319.484,A -85,B 0,C 180,E1 -6968.854,E2 -6968.854} C_VEL
LIN {X 0,Y 481.669,Z 319.49,A -85,B 0,C 180,E1 -6972.157,E2 -6972.157} C_VEL
LIN {X 0,Y 481.655,Z 319.488,A -85,B 0,C 180,E1 -6974.456,E2 -6974.456} C_VEL
LIN {X 0,Y 481.622,Z 319.49,A -85,B 0,C 180,E1 -6977.836,E2 -6977.836} C_VEL
LIN {X 0,Y 481.661,Z 319.486,A -85,B 0,C 180,E1 -6981.14,E2 -6981.14} C_VEL
LIN {X 0,Y 481.661,Z 319.487,A -85,B 0,C 180,E1 -6984.794,E2 -6984.794} C_VEL
LIN {X 0,Y 481.664,Z 319.488,A -85,B 0,C 180,E1 -6987.325,E2 -6987.325} C_VEL
LIN {X 0,Y 481.657,Z 319.487,A -85,B 0,C 180,E1 -6990.257,E2 -6990.257} C_VEL
LIN {X 0,Y 481.673,Z 319.483,A -85,B 0,C 180,E1 -6993.108,E2 -6993.108} C_VEL
LIN {X 0,Y 481.65,Z 319.489,A -85,B 0,C 180,E1 -6995.885,E2 -6995.885} C_VEL
LIN {X 0,Y 481.693,Z 319.484,A -85,B 0,C 180,E1 -6999.027,E2 -6999.027} C_VEL
LIN {X 0,Y 481.696,Z 319.483,A -85,B 0,C 180,E1 -7002.158,E2 -7002.158} C_VEL
LIN {X 0,Y 481.728,Z 319.479,A -85,B 0,C 180,E1 -7004.775,E2 -7004.775} C_VEL
LIN {X 0,Y 481.74,Z 319.479,A -85,B 0,C 180,E1 -7008.215,E2 -7008.215} C_VEL
LIN {X 0,Y 481.753,Z 319.479,A -85,B 0,C 180,E1 -7011.612,E2 -7011.612} C_VEL
LIN {X 0,Y 481.822,Z 319.467,A -85,B 0,C 180,E1 -7014.14,E2 -7014.14} C_VEL
LIN {X 0,Y 481.918,Z 319.455,A -85,B 0,C 180,E1 -7017.493,E2 -7017.493} C_VEL
LIN {X 0,Y 481.926,Z 319.456,A -85,B 0,C 180,E1 -7020,E2 -7020} C_VEL
LIN {X 0,Y 481.917,Z 319.452,A -85,B 0,C 180,E1 -7022.508,E2 -7022.508} C_VEL
LIN {X 0,Y 481.815,Z 319.467,A -85,B 0,C 180,E1 -7025.86,E2 -7025.86} C_VEL
LIN {X 0,Y 481.753,Z 319.476,A -85,B 0,C 180,E1 -7028.389,E2 -7028.389} C_VEL
LIN {X 0,Y 481.74,Z 319.48,A -85,B 0,C 180,E1 -7031.785,E2 -7031.785} C_VEL
LIN {X 0,Y 481.729,Z 319.481,A -85,B 0,C 180,E1 -7035.225,E2 -7035.225} C_VEL
LIN {X 0,Y 481.703,Z 319.483,A -85,B 0,C 180,E1 -7038.722,E2 -7038.722} C_VEL
LIN {X 0,Y 481.638,Z 319.49,A -85,B 0,C 180,E1 -7041.395,E2 -7041.395} C_VEL
LIN {X 0,Y 481.65,Z 319.489,A -85,B 0,C 180,E1 -7044.115,E2 -7044.115} C_VEL
LIN {X 0,Y 481.681,Z 319.487,A -85,B 0,C 180,E1 -7047.127,E2 -7047.127} C_VEL
LIN {X 0,Y 481.657,Z 319.485,A -85,B 0,C 180,E1 -7049.743,E2 -7049.743} C_VEL
LIN {X 0,Y 481.664,Z 319.49,A -85,B 0,C 180,E1 -7052.675,E2 -7052.675} C_VEL
LIN {X 0,Y 481.636,Z 319.491,A -85,B 0,C 180,E1 -7055.71,E2 -7055.71} C_VEL
LIN {X 0,Y 481.661,Z 319.488,A -85,B 0,C 180,E1 -7058.86,E2 -7058.86} C_VEL
LIN {X 0,Y 481.618,Z 319.492,A -85,B 0,C 180,E1 -7062.164,E2 -7062.164} C_VEL
LIN {X 0,Y 481.649,Z 319.486,A -85,B 0,C 180,E1 -7065.543,E2 -7065.543} C_VEL
LIN {X 0,Y 481.664,Z 319.486,A -85,B 0,C 180,E1 -7068.961,E2 -7068.961} C_VEL
LIN {X 0,Y 481.693,Z 319.484,A -85,B 0,C 180,E1 -7071.144,E2 -7071.144} C_VEL
LIN {X 0,Y 481.538,Z 319.504,A -85,B 0,C 180,E1 -7074.283,E2 -7074.283} C_VEL
LIN {X 0,Y 481.534,Z 319.793,A -85,B 0,C 180,E1 -7074.818,E2 -7074.818} C_VEL
LIN {X 0,Y 481.519,Z 323.266,A -85,B 0,C 180,E1 -7077.315,E2 -7077.315} C_VEL
LIN {X 0,Y 481.407,Z 327.436,A -85,B 0,C 180,E1 -7080.242,E2 -7080.242} C_VEL
LIN {X 0,Y 481.28,Z 331.573,A -85,B 0,C 180,E1 -7083.085,E2 -7083.085} C_VEL
LIN {X 0,Y 481.229,Z 335.702,A -85,B 0,C 180,E1 -7085.864,E2 -7085.864} C_VEL
LIN {X 0,Y 481.108,Z 338.533,A -85,B 0,C 180,E1 -7087.741,E2 -7087.741} C_VEL
LIN {X 0,Y 480.398,Z 339.642,A -85,B 0,C 180,E1 -7088.428,E2 -7088.428} C_VEL
LIN {X 0,Y 477.5,Z 341.618,A -85,B 0,C 180,E1 -7089.538,E2 -7089.538} C_VEL
LIN {X 0,Y 475.075,Z 343.224,A -85,B 0,C 180,E1 -7090.432,E2 -7090.432} C_VEL
LIN {X 0,Y 474.043,Z 344.395,A -85,B 0,C 180,E1 -7091.124,E2 -7091.124} C_VEL
LIN {X 0,Y 473.962,Z 344.77,A -85,B 0,C 180,E1 -7091.359,E2 -7091.359} C_VEL
LIN {X 0,Y 473.987,Z 350.656,A -85,B 0,C 180,E1 -7094.914,E2 -7094.914} C_VEL
LIN {X 0,Y 476.654,Z 363.785,A -85,B 0,C 180,E1 -7095.376,E2 -7095.376} C_VEL
LIN {X 0,Y 477.067,Z 368.123,A -85,B 0,C 180,E1 -7095.552,E2 -7095.552} C_VEL
LIN {X 0,Y 476.701,Z 380.67,A -85,B 0,C 180,E1 -7096.139,E2 -7096.139} C_VEL
LIN {X 0,Y 476.257,Z 392.164,A -85,B 0,C 180,E1 -7096.851,E2 -7096.851} C_VEL
LIN {X 0,Y 475.877,Z 403.37,A -85,B 0,C 180,E1 -7097.744,E2 -7097.744} C_VEL
LIN {X 0,Y 475.416,Z 413.095,A -85,B 0,C 180,E1 -7098.705,E2 -7098.705} C_VEL
LIN {X 0,Y 474.973,Z 421.94,A -85,B 0,C 180,E1 -7099.773,E2 -7099.773} C_VEL
LIN {X 0,Y 474.573,Z 430.569,A -85,B 0,C 180,E1 -7101.055,E2 -7101.055} C_VEL
LIN {X 0,Y 474.225,Z 437.447,A -85,B 0,C 180,E1 -7102.336,E2 -7102.336} C_VEL
LIN {X 0,Y 474.071,Z 442.985,A -85,B 0,C 180,E1 -7103.626,E2 -7103.626} C_VEL
LIN {X 0,Y 473.854,Z 447.275,A -85,B 0,C 180,E1 -7104.895,E2 -7104.895} C_VEL
LIN {X 0,Y 473.877,Z 449.559,A -85,B 0,C 180,E1 -7105.748,E2 -7105.748} C_VEL
LIN {X 0,Y 473.842,Z 451.42,A -85,B 0,C 180,E1 -7106.599,E2 -7106.599} C_VEL
LIN {X 0,Y 473.763,Z 452.825,A -85,B 0,C 180,E1 -7107.45,E2 -7107.45} C_VEL
LIN {X 0,Y 473.689,Z 454.438,A -85,B 0,C 180,E1 -7109.15,E2 -7109.15} C_VEL
LIN {X 0,Y 473.67,Z 454.674,A -85,B 0,C 180,E1 -7110,E2 -7110} C_VEL
LIN {X 0,Y 473.689,Z 454.488,A -85,B 0,C 180,E1 -7110.85,E2 -7110.85} C_VEL
LIN {X 0,Y 473.764,Z 452.939,A -85,B 0,C 180,E1 -7112.551,E2 -7112.551} C_VEL
LIN {X 0,Y 473.842,Z 451.584,A -85,B 0,C 180,E1 -7113.402,E2 -7113.402} C_VEL
LIN {X 0,Y 473.83,Z 448.724,A -85,B 0,C 180,E1 -7114.68,E2 -7114.68} C_VEL
LIN {X 0,Y 474.075,Z 444.839,A -85,B 0,C 180,E1 -7115.957,E2 -7115.957} C_VEL
LIN {X 0,Y 474.147,Z 439.834,A -85,B 0,C 180,E1 -7117.238,E2 -7117.238} C_VEL
LIN {X 0,Y 474.422,Z 433.53,A -85,B 0,C 180,E1 -7118.519,E2 -7118.519} C_VEL
LIN {X 0,Y 474.763,Z 425.637,A -85,B 0,C 180,E1 -7119.802,E2 -7119.802} C_VEL
LIN {X 0,Y 475.138,Z 417.589,A -85,B 0,C 180,E1 -7120.871,E2 -7120.871} C_VEL
LIN {X 0,Y 475.66,Z 407.765,A -85,B 0,C 180,E1 -7121.938,E2 -7121.938} C_VEL
LIN {X 0,Y 476.081,Z 396.617,A -85,B 0,C 180,E1 -7122.91,E2 -7122.91} C_VEL
LIN {X 0,Y 476.46,Z 385.895,A -85,B 0,C 180,E1 -7123.651,E2 -7123.651} C_VEL
LIN {X 0,Y 476.923,Z 373.934,A -85,B 0,C 180,E1 -7124.29,E2 -7124.29} C_VEL
LIN {X 0,Y 476.885,Z 365.198,A -85,B 0,C 180,E1 -7124.657,E2 -7124.657} C_VEL
LIN {X 0,Y 474.377,Z 352.651,A -85,B 0,C 180,E1 -7125.117,E2 -7125.117} C_VEL
LIN {X 0,Y 473.973,Z 350.438,A -85,B 0,C 180,E1 -7125.196,E2 -7125.196} C_VEL
LIN {X 0,Y 473.97,Z 344.31,A -85,B 0,C 180,E1 -7129.039,E2 -7129.039} C_VEL
LIN {X 0,Y 474.042,Z 340.107,A -85,B 0,C 180,E1 -7131.755,E2 -7131.755} C_VEL
LIN {X 0,Y 474.135,Z 335.994,A -85,B 0,C 180,E1 -7134.522,E2 -7134.522} C_VEL
LIN {X 0,Y 474.24,Z 331.86,A -85,B 0,C 180,E1 -7137.349,E2 -7137.349} C_VEL
LIN {X 0,Y 474.367,Z 327.692,A -85,B 0,C 180,E1 -7140.247,E2 -7140.247} C_VEL
LIN {X 0,Y 474.499,Z 323.49,A -85,B 0,C 180,E1 -7143.231,E2 -7143.231} C_VEL
LIN {X 0,Y 474.52,Z 320.464,A -85,B 0,C 180,E1 -7145.453,E2 -7145.453} C_VEL
LIN {X 0,Y 474.609,Z 320.368,A -85,B 0,C 180,E1 -7148.457,E2 -7148.457} C_VEL
LIN {X 0,Y 474.62,Z 320.366,A -85,B 0,C 180,E1 -7151.785,E2 -7151.785} C_VEL
LIN {X 0,Y 474.615,Z 320.362,A -85,B 0,C 180,E1 -7154.702,E2 -7154.702} C_VEL
LIN {X 0,Y 474.574,Z 320.37,A -85,B 0,C 180,E1 -7157.769,E2 -7157.769} C_VEL
LIN {X 0,Y 474.619,Z 320.364,A -85,B 0,C 180,E1 -7160.451,E2 -7160.451} C_VEL
LIN {X 0,Y 474.59,Z 320.37,A -85,B 0,C 180,E1 -7163.676,E2 -7163.676} C_VEL
LIN {X 0,Y 474.64,Z 320.361,A -85,B 0,C 180,E1 -7166.78,E2 -7166.78} C_VEL
LIN {X 0,Y 474.593,Z 320.366,A -85,B 0,C 180,E1 -7169.769,E2 -7169.769} C_VEL
LIN {X 0,Y 474.633,Z 320.364,A -85,B 0,C 180,E1 -7172.676,E2 -7172.676} C_VEL
LIN {X 0,Y 474.623,Z 320.365,A -85,B 0,C 180,E1 -7175.505,E2 -7175.505} C_VEL
LIN {X 0,Y 474.63,Z 320.363,A -85,B 0,C 180,E1 -7178.883,E2 -7178.883} C_VEL
LIN {X 0,Y 474.651,Z 320.359,A -85,B 0,C 180,E1 -7181.884,E2 -7181.884} C_VEL
LIN {X 0,Y 474.694,Z 320.357,A -85,B 0,C 180,E1 -7184.544,E2 -7184.544} C_VEL
LIN {X 0,Y 474.699,Z 320.355,A -85,B 0,C 180,E1 -7188.037,E2 -7188.037} C_VEL
LIN {X 0,Y 474.723,Z 320.352,A -85,B 0,C 180,E1 -7191.486,E2 -7191.486} C_VEL
LIN {X 0,Y 474.777,Z 320.344,A -85,B 0,C 180,E1 -7194.052,E2 -7194.052} C_VEL
LIN {X 0,Y 474.889,Z 320.328,A -85,B 0,C 180,E1 -7197.455,E2 -7197.455} C_VEL
LIN {X 0,Y 474.9,Z 320.331,A -85,B 0,C 180,E1 -7200,E2 -7200} C_VEL
LIN {X 0,Y 474.888,Z 320.331,A -85,B 0,C 180,E1 -7202.545,E2 -7202.545} C_VEL
LIN {X 0,Y 474.777,Z 320.345,A -85,B 0,C 180,E1 -7205.948,E2 -7205.948} C_VEL
LIN {X 0,Y 474.724,Z 320.353,A -85,B 0,C 180,E1 -7208.514,E2 -7208.514} C_VEL
LIN {X 0,Y 474.699,Z 320.357,A -85,B 0,C 180,E1 -7211.963,E2 -7211.963} C_VEL
LIN {X 0,Y 474.675,Z 320.36,A -85,B 0,C 180,E1 -7215.768,E2 -7215.768} C_VEL
LIN {X 0,Y 474.661,Z 320.36,A -85,B 0,C 180,E1 -7219.01,E2 -7219.01} C_VEL
LIN {X 0,Y 474.587,Z 320.369,A -85,B 0,C 180,E1 -7221.729,E2 -7221.729} C_VEL
LIN {X 0,Y 474.633,Z 320.361,A -85,B 0,C 180,E1 -7224.494,E2 -7224.494} C_VEL
LIN {X 0,Y 474.633,Z 320.364,A -85,B 0,C 180,E1 -7227.324,E2 -7227.324} C_VEL
LIN {X 0,Y 474.597,Z 320.367,A -85,B 0,C 180,E1 -7230.81,E2 -7230.81} C_VEL
LIN {X 0,Y 474.636,Z 320.364,A -85,B 0,C 180,E1 -7233.984,E2 -7233.984} C_VEL
LIN {X 0,Y 474.571,Z 320.37,A -85,B 0,C 180,E1 -7236.9,E2 -7236.9} C_VEL
LIN {X 0,Y 474.602,Z 320.367,A -85,B 0,C 180,E1 -7239.645,E2 -7239.645} C_VEL
LIN {X 0,Y 474.566,Z 320.374,A -85,B 0,C 180,E1 -7242.94,E2 -7242.94} C_VEL
LIN {X 0,Y 474.605,Z 320.368,A -85,B 0,C 180,E1 -7245.895,E2 -7245.895} C_VEL
LIN {X 0,Y 474.627,Z 320.364,A -85,B 0,C 180,E1 -7249.041,E2 -7249.041} C_VEL
LIN {X 0,Y 474.675,Z 320.482,A -85,B 0,C 180,E1 -7251.074,E2 -7251.074} C_VEL
LIN {X 0,Y 475.483,Z 325.922,A -85,B 0,C 180,E1 -7253.756,E2 -7253.756} C_VEL
LIN {X 0,Y 475.515,Z 330.473,A -85,B 0,C 180,E1 -7255.86,E2 -7255.86} C_VEL
LIN {X 0,Y 475.232,Z 337.708,A -85,B 0,C 180,E1 -7259.064,E2 -7259.064} C_VEL
LIN {X 0,Y 475.002,Z 345.076,A -85,B 0,C 180,E1 -7262.221,E2 -7262.221} C_VEL
LIN {X 0,Y 474.69,Z 352.959,A -85,B 0,C 180,E1 -7265.509,E2 -7265.509} C_VEL
LIN {X 0,Y 474.504,Z 359.798,A -85,B 0,C 180,E1 -7268.267,E2 -7268.267} C_VEL
LIN {X 0,Y 474.345,Z 366.615,A -85,B 0,C 180,E1 -7270.976,E2 -7270.976} C_VEL
LIN {X 0,Y 474.178,Z 376.241,A -85,B 0,C 180,E1 -7274.747,E2 -7274.747} C_VEL
LIN {X 0,Y 474.141,Z 376.452,A -85,B 0,C 180,E1 -7274.828,E2 -7274.828} C_VEL
LIN {X 0,Y 476.551,Z 390.308,A -85,B 0,C 180,E1 -7275.276,E2 -7275.276} C_VEL
LIN {X 0,Y 477.063,Z 394.499,A -85,B 0,C 180,E1 -7275.442,E2 -7275.442} C_VEL
LIN {X 0,Y 476.605,Z 407.501,A -85,B 0,C 180,E1 -7276.027,E2 -7276.027} C_VEL
LIN {X 0,Y 476.185,Z 418.675,A -85,B 0,C 180,E1 -7276.7,E2 -7276.7} C_VEL
LIN {X 0,Y 475.781,Z 429.482,A -85,B 0,C 180,E1 -7277.524,E2 -7277.524} C_VEL
LIN {X 0,Y 475.335,Z 439.644,A -85,B 0,C 180,E1 -7278.486,E2 -7278.486} C_VEL
LIN {X 0,Y 474.878,Z 448.784,A -85,B 0,C 180,E1 -7279.555,E2 -7279.555} C_VEL
LIN {X 0,Y 474.482,Z 457.686,A -85,B 0,C 180,E1 -7280.838,E2 -7280.838} C_VEL
LIN {X 0,Y 474.153,Z 464.847,A -85,B 0,C 180,E1 -7282.119,E2 -7282.119} C_VEL
LIN {X 0,Y 473.977,Z 470.719,A -85,B 0,C 180,E1 -7283.443,E2 -7283.443} C_VEL
LIN {X 0,Y 473.846,Z 475.676,A -85,B 0,C 180,E1 -7284.894,E2 -7284.894} C_VEL
LIN {X 0,Y 473.752,Z 477.957,A -85,B 0,C 180,E1 -7285.746,E2 -7285.746} C_VEL
LIN {X 0,Y 473.8,Z 479.806,A -85,B 0,C 180,E1 -7286.598,E2 -7286.598} C_VEL
LIN {X 0,Y 473.695,Z 482.182,A -85,B 0,C 180,E1 -7288.299,E2 -7288.299} C_VEL
LIN {X 0,Y 473.688,Z 482.785,A -85,B 0,C 180,E1 -7289.15,E2 -7289.15} C_VEL
LIN {X 0,Y 473.669,Z 483,A -85,B 0,C 180,E1 -7290,E2 -7290} C_VEL
LIN {X 0,Y 473.688,Z 482.786,A -85,B 0,C 180,E1 -7290.85,E2 -7290.85} C_VEL
LIN {X 0,Y 473.724,Z 481.196,A -85,B 0,C 180,E1 -7292.55,E2 -7292.55} C_VEL
LIN {X 0,Y 473.799,Z 479.811,A -85,B 0,C 180,E1 -7293.401,E2 -7293.401} C_VEL
LIN {X 0,Y 473.775,Z 476.896,A -85,B 0,C 180,E1 -7294.679,E2 -7294.679} C_VEL
LIN {X 0,Y 473.942,Z 472.95,A -85,B 0,C 180,E1 -7295.958,E2 -7295.958} C_VEL
LIN {X 0,Y 474.049,Z 466.878,A -85,B 0,C 180,E1 -7297.453,E2 -7297.453} C_VEL
LIN {X 0,Y 474.377,Z 460.238,A -85,B 0,C 180,E1 -7298.734,E2 -7298.734} C_VEL
LIN {X 0,Y 474.751,Z 451.996,A -85,B 0,C 180,E1 -7300.017,E2 -7300.017} C_VEL
LIN {X 0,Y 475.101,Z 443.545,A -85,B 0,C 180,E1 -7301.087,E2 -7301.087} C_VEL
LIN {X 0,Y 475.62,Z 433.119,A -85,B 0,C 180,E1 -7302.153,E2 -7302.153} C_VEL
LIN {X 0,Y 476.027,Z 422.048,A -85,B 0,C 180,E1 -7303.065,E2 -7303.065} C_VEL
LIN {X 0,Y 476.473,Z 411.414,A -85,B 0,C 180,E1 -7303.759,E2 -7303.759} C_VEL
LIN {X 0,Y 476.894,Z 399.78,A -85,B 0,C 180,E1 -7304.345,E2 -7304.345} C_VEL
LIN {X 0,Y 476.892,Z 392.606,A -85,B 0,C 180,E1 -7304.631,E2 -7304.631} C_VEL
LIN {X 0,Y 474.74,Z 379.935,A -85,B 0,C 180,E1 -7305.072,E2 -7305.072} C_VEL
LIN {X 0,Y 474.139,Z 376.45,A -85,B 0,C 180,E1 -7305.171,E2 -7305.171} C_VEL
LIN {X 0,Y 474.276,Z 367.953,A -85,B 0,C 180,E1 -7308.49,E2 -7308.49} C_VEL
LIN {X 0,Y 474.453,Z 361.453,A -85,B 0,C 180,E1 -7311.059,E2 -7311.059} C_VEL
LIN {X 0,Y 474.667,Z 354.066,A -85,B 0,C 180,E1 -7314.026,E2 -7314.026} C_VEL
LIN {X 0,Y 474.936,Z 345.995,A -85,B 0,C 180,E1 -7317.393,E2 -7317.393} C_VEL
LIN {X 0,Y 475.192,Z 339.433,A -85,B 0,C 180,E1 -7320.188,E2 -7320.188} C_VEL
LIN {X 0,Y 475.419,Z 332.657,A -85,B 0,C 180,E1 -7323.158,E2 -7323.158} C_VEL
LIN {X 0,Y 475.596,Z 327.2,A -85,B 0,C 180,E1 -7325.634,E2 -7325.634} C_VEL
LIN {X 0,Y 475.039,Z 322.653,A -85,B 0,C 180,E1 -7327.832,E2 -7327.832} C_VEL
LIN {X 0,Y 474.665,Z 320.362,A -85,B 0,C 180,E1 -7328.995,E2 -7328.995} C_VEL
LIN {X 0,Y 474.644,Z 320.365,A -85,B 0,C 180,E1 -7332.239,E2 -7332.239} C_VEL
LIN {X 0,Y 474.615,Z 320.369,A -85,B 0,C 180,E1 -7335.296,E2 -7335.296} C_VEL
LIN {X 0,Y 474.597,Z 320.365,A -85,B 0,C 180,E1 -7338.212,E2 -7338.212} C_VEL
LIN {X 0,Y 474.603,Z 320.365,A -85,B 0,C 180,E1 -7341.542,E2 -7341.542} C_VEL
LIN {X 0,Y 474.623,Z 320.364,A -85,B 0,C 180,E1 -7344.725,E2 -7344.725} C_VEL
LIN {X 0,Y 474.627,Z 320.364,A -85,B 0,C 180,E1 -7347.787,E2 -7347.787} C_VEL
LIN {X 0,Y 474.589,Z 320.37,A -85,B 0,C 180,E1 -7350.89,E2 -7350.89} C_VEL
LIN {X 0,Y 474.605,Z 320.363,A -85,B 0,C 180,E1 -7353.625,E2 -7353.625} C_VEL
LIN {X 0,Y 474.625,Z 320.363,A -85,B 0,C 180,E1 -7356.641,E2 -7356.641} C_VEL
LIN {X 0,Y 474.647,Z 320.361,A -85,B 0,C 180,E1 -7360.089,E2 -7360.089} C_VEL
LIN {X 0,Y 474.638,Z 320.363,A -85,B 0,C 180,E1 -7362.774,E2 -7362.774} C_VEL
LIN {X 0,Y 474.629,Z 320.362,A -85,B 0,C 180,E1 -7365.42,E2 -7365.42} C_VEL
LIN {X 0,Y 474.694,Z 320.359,A -85,B 0,C 180,E1 -7368.037,E2 -7368.037} C_VEL
LIN {X 0,Y 474.718,Z 320.354,A -85,B 0,C 180,E1 -7371.486,E2 -7371.486} C_VEL
LIN {X 0,Y 474.782,Z 320.344,A -85,B 0,C 180,E1 -7374.052,E2 -7374.052} C_VEL
LIN {X 0,Y 474.884,Z 320.331,A -85,B 0,C 180,E1 -7377.455,E2 -7377.455} C_VEL
LIN {X 0,Y 474.896,Z 320.332,A -85,B 0,C 180,E1 -7380,E2 -7380} C_VEL
LIN {X 0,Y 474.884,Z 320.328,A -85,B 0,C 180,E1 -7382.545,E2 -7382.545} C_VEL
LIN {X 0,Y 474.776,Z 320.344,A -85,B 0,C 180,E1 -7385.948,E2 -7385.948} C_VEL
LIN {X 0,Y 474.718,Z 320.352,A -85,B 0,C 180,E1 -7388.514,E2 -7388.514} C_VEL
LIN {X 0,Y 474.693,Z 320.356,A -85,B 0,C 180,E1 -7391.963,E2 -7391.963} C_VEL
LIN {X 0,Y 474.67,Z 320.357,A -85,B 0,C 180,E1 -7395.768,E2 -7395.768} C_VEL
LIN {X 0,Y 474.656,Z 320.363,A -85,B 0,C 180,E1 -7399.011,E2 -7399.011} C_VEL
LIN {X 0,Y 474.581,Z 320.37,A -85,B 0,C 180,E1 -7401.729,E2 -7401.729} C_VEL
LIN {X 0,Y 474.629,Z 320.364,A -85,B 0,C 180,E1 -7404.495,E2 -7404.495} C_VEL
LIN {X 0,Y 474.628,Z 320.366,A -85,B 0,C 180,E1 -7407.325,E2 -7407.325} C_VEL
LIN {X 0,Y 474.593,Z 320.371,A -85,B 0,C 180,E1 -7410.81,E2 -7410.81} C_VEL
LIN {X 0,Y 474.631,Z 320.362,A -85,B 0,C 180,E1 -7413.985,E2 -7413.985} C_VEL
LIN {X 0,Y 474.568,Z 320.371,A -85,B 0,C 180,E1 -7416.901,E2 -7416.901} C_VEL
LIN {X 0,Y 474.599,Z 320.367,A -85,B 0,C 180,E1 -7419.645,E2 -7419.645} C_VEL
LIN {X 0,Y 474.568,Z 320.372,A -85,B 0,C 180,E1 -7422.94,E2 -7422.94} C_VEL
LIN {X 0,Y 474.601,Z 320.365,A -85,B 0,C 180,E1 -7425.896,E2 -7425.896} C_VEL
LIN {X 0,Y 474.637,Z 320.362,A -85,B 0,C 180,E1 -7429.04,E2 -7429.04} C_VEL
LIN {X 0,Y 474.61,Z 320.367,A -85,B 0,C 180,E1 -7431.705,E2 -7431.705} C_VEL
LIN {X 0,Y 474.508,Z 320.559,A -85,B 0,C 180,E1 -7434.717,E2 -7434.717} C_VEL
LIN {X 0,Y 474.498,Z 323.374,A -85,B 0,C 180,E1 -7436.77,E2 -7436.77} C_VEL
LIN {X 0,Y 474.37,Z 327.555,A -85,B 0,C 180,E1 -7439.754,E2 -7439.754} C_VEL
LIN {X 0,Y 474.236,Z 331.881,A -85,B 0,C 180,E1 -7442.771,E2 -7442.771} C_VEL
LIN {X 0,Y 474.17,Z 335.845,A -85,B 0,C 180,E1 -7445.481,E2 -7445.481} C_VEL
LIN {X 0,Y 474.041,Z 339.968,A -85,B 0,C 180,E1 -7448.246,E2 -7448.246} C_VEL
LIN {X 0,Y 473.962,Z 344.77,A -85,B 0,C 180,E1 -7451.359,E2 -7451.359} C_VEL
LIN {X 0,Y 473.276,Z 345.56,A -85,B 0,C 180,E1 -7451.822,E2 -7451.822} C_VEL
LIN {X 0,Y 470.381,Z 346.951,A -85,B 0,C 180,E1 -7452.541,E2 -7452.541} C_VEL
LIN {X 0,Y 467.481,Z 348.356,A -85,B 0,C 180,E1 -7453.267,E2 -7453.267} C_VEL
LIN {X 0,Y 466.806,Z 349.167,A -85,B 0,C 180,E1 -7453.739,E2 -7453.739} C_VEL
LIN {X 0,Y 466.906,Z 350.65,A -85,B 0,C 180,E1 -7454.666,E2 -7454.666} C_VEL
LIN {X 0,Y 469.853,Z 365.149,A -85,B 0,C 180,E1 -7455.201,E2 -7455.201} C_VEL
LIN {X 0,Y 470.186,Z 369.647,A -85,B 0,C 180,E1 -7455.391,E2 -7455.391} C_VEL
LIN {X 0,Y 469.82,Z 380.895,A -85,B 0,C 180,E1 -7455.932,E2 -7455.932} C_VEL
LIN {X 0,Y 469.325,Z 392.857,A -85,B 0,C 180,E1 -7456.686,E2 -7456.686} C_VEL
LIN {X 0,Y 468.933,Z 403.591,A -85,B 0,C 180,E1 -7457.559,E2 -7457.559} C_VEL
LIN {X 0,Y 468.462,Z 413.315,A -85,B 0,C 180,E1 -7458.535,E2 -7458.535} C_VEL
LIN {X 0,Y 467.991,Z 422.159,A -85,B 0,C 180,E1 -7459.619,E2 -7459.619} C_VEL
LIN {X 0,Y 467.555,Z 430.787,A -85,B 0,C 180,E1 -7460.92,E2 -7460.92} C_VEL
LIN {X 0,Y 467.2,Z 437.664,A -85,B 0,C 180,E1 -7462.22,E2 -7462.22} C_VEL
LIN {X 0,Y 467.007,Z 443.529,A -85,B 0,C 180,E1 -7463.618,E2 -7463.618} C_VEL
LIN {X 0,Y 466.798,Z 447.491,A -85,B 0,C 180,E1 -7464.818,E2 -7464.818} C_VEL
LIN {X 0,Y 466.781,Z 449.776,A -85,B 0,C 180,E1 -7465.683,E2 -7465.683} C_VEL
LIN {X 0,Y 466.775,Z 451.636,A -85,B 0,C 180,E1 -7466.548,E2 -7466.548} C_VEL
LIN {X 0,Y 466.684,Z 453.04,A -85,B 0,C 180,E1 -7467.411,E2 -7467.411} C_VEL
LIN {X 0,Y 466.62,Z 454.653,A -85,B 0,C 180,E1 -7469.137,E2 -7469.137} C_VEL
LIN {X 0,Y 466.599,Z 454.889,A -85,B 0,C 180,E1 -7470,E2 -7470} C_VEL
LIN {X 0,Y 466.62,Z 454.702,A -85,B 0,C 180,E1 -7470.863,E2 -7470.863} C_VEL
LIN {X 0,Y 466.684,Z 453.153,A -85,B 0,C 180,E1 -7472.59,E2 -7472.59} C_VEL
LIN {X 0,Y 466.774,Z 451.798,A -85,B 0,C 180,E1 -7473.453,E2 -7473.453} C_VEL
LIN {X 0,Y 466.748,Z 448.939,A -85,B 0,C 180,E1 -7474.751,E2 -7474.751} C_VEL
LIN {X 0,Y 467.019,Z 445.053,A -85,B 0,C 180,E1 -7476.047,E2 -7476.047} C_VEL
LIN {X 0,Y 467.101,Z 440.048,A -85,B 0,C 180,E1 -7477.348,E2 -7477.348} C_VEL
LIN {X 0,Y 467.409,Z 433.743,A -85,B 0,C 180,E1 -7478.648,E2 -7478.648} C_VEL
LIN {X 0,Y 467.758,Z 425.849,A -85,B 0,C 180,E1 -7479.95,E2 -7479.95} C_VEL
LIN {X 0,Y 468.143,Z 417.802,A -85,B 0,C 180,E1 -7481.035,E2 -7481.035} C_VEL
LIN {X 0,Y 468.728,Z 407.975,A -85,B 0,C 180,E1 -7482.117,E2 -7482.117} C_VEL
LIN {X 0,Y 469.164,Z 396.794,A -85,B 0,C 180,E1 -7483.106,E2 -7483.106} C_VEL
LIN {X 0,Y 469.562,Z 386.103,A -85,B 0,C 180,E1 -7483.856,E2 -7483.856} C_VEL
LIN {X 0,Y 470.065,Z 374.139,A -85,B 0,C 180,E1 -7484.503,E2 -7484.503} C_VEL
LIN {X 0,Y 470.056,Z 366.405,A -85,B 0,C 180,E1 -7484.838,E2 -7484.838} C_VEL
LIN {X 0,Y 467.533,Z 353.792,A -85,B 0,C 180,E1 -7485.32,E2 -7485.32} C_VEL
LIN {X 0,Y 466.882,Z 350.641,A -85,B 0,C 180,E1 -7485.432,E2 -7485.432} C_VEL
LIN {X 0,Y 466.886,Z 345.783,A -85,B 0,C 180,E1 -7488.497,E2 -7488.497} C_VEL
LIN {X 0,Y 466.979,Z 341.676,A -85,B 0,C 180,E1 -7491.174,E2 -7491.174} C_VEL
LIN {X 0,Y 467.058,Z 337.523,A -85,B 0,C 180,E1 -7493.971,E2 -7493.971} C_VEL
LIN {X 0,Y 467.151,Z 333.387,A -85,B 0,C 180,E1 -7496.829,E2 -7496.829} C_VEL
LIN {X 0,Y 467.283,Z 329.208,A -85,B 0,C 180,E1 -7499.757,E2 -7499.757} C_VEL
LIN {X 0,Y 467.42,Z 325.007,A -85,B 0,C 180,E1 -7502.771,E2 -7502.771} C_VEL
LIN {X 0,Y 467.494,Z 322.204,A -85,B 0,C 180,E1 -7504.838,E2 -7504.838} C_VEL
LIN {X 0,Y 467.489,Z 321.253,A -85,B 0,C 180,E1 -7505.895,E2 -7505.895} C_VEL
LIN {X 0,Y 467.558,Z 321.247,A -85,B 0,C 180,E1 -7508.59,E2 -7508.59} C_VEL
LIN {X 0,Y 467.576,Z 321.241,A -85,B 0,C 180,E1 -7511.402,E2 -7511.402} C_VEL
LIN {X 0,Y 467.551,Z 321.247,A -85,B 0,C 180,E1 -7513.82,E2 -7513.82} C_VEL
LIN {X 0,Y 467.543,Z 321.244,A -85,B 0,C 180,E1 -7516.254,E2 -7516.254} C_VEL
LIN {X 0,Y 467.555,Z 321.244,A -85,B 0,C 180,E1 -7519.733,E2 -7519.733} C_VEL
LIN {X 0,Y 467.547,Z 321.247,A -85,B 0,C 180,E1 -7522.813,E2 -7522.813} C_VEL
LIN {X 0,Y 467.584,Z 321.24,A -85,B 0,C 180,E1 -7526.211,E2 -7526.211} C_VEL
LIN {X 0,Y 467.563,Z 321.246,A -85,B 0,C 180,E1 -7529.265,E2 -7529.265} C_VEL
LIN {X 0,Y 467.57,Z 321.242,A -85,B 0,C 180,E1 -7532.475,E2 -7532.475} C_VEL
LIN {X 0,Y 467.564,Z 321.244,A -85,B 0,C 180,E1 -7535.11,E2 -7535.11} C_VEL
LIN {X 0,Y 467.53,Z 321.247,A -85,B 0,C 180,E1 -7537.926,E2 -7537.926} C_VEL
LIN {X 0,Y 467.62,Z 321.236,A -85,B 0,C 180,E1 -7540.692,E2 -7540.692} C_VEL
LIN {X 0,Y 467.645,Z 321.231,A -85,B 0,C 180,E1 -7544.115,E2 -7544.115} C_VEL
LIN {X 0,Y 467.651,Z 321.232,A -85,B 0,C 180,E1 -7547.854,E2 -7547.854} C_VEL
LIN {X 0,Y 467.677,Z 321.23,A -85,B 0,C 180,E1 -7551.357,E2 -7551.357} C_VEL
LIN {X 0,Y 467.741,Z 321.221,A -85,B 0,C 180,E1 -7553.963,E2 -7553.963} C_VEL
LIN {X 0,Y 467.854,Z 321.204,A -85,B 0,C 180,E1 -7557.417,E2 -7557.417} C_VEL
LIN {X 0,Y 467.87,Z 321.206,A -85,B 0,C 180,E1 -7560,E2 -7560} C_VEL
LIN {X 0,Y 467.853,Z 321.207,A -85,B 0,C 180,E1 -7562.583,E2 -7562.583} C_VEL
LIN {X 0,Y 467.741,Z 321.221,A -85,B 0,C 180,E1 -7566.037,E2 -7566.037} C_VEL
LIN {X 0,Y 467.678,Z 321.23,A -85,B 0,C 180,E1 -7568.643,E2 -7568.643} C_VEL
LIN {X 0,Y 467.651,Z 321.235,A -85,B 0,C 180,E1 -7572.146,E2 -7572.146} C_VEL
LIN {X 0,Y 467.644,Z 321.234,A -85,B 0,C 180,E1 -7575.885,E2 -7575.885} C_VEL
LIN {X 0,Y 467.62,Z 321.238,A -85,B 0,C 180,E1 -7579.308,E2 -7579.308} C_VEL
LIN {X 0,Y 467.533,Z 321.25,A -85,B 0,C 180,E1 -7582.074,E2 -7582.074} C_VEL
LIN {X 0,Y 467.579,Z 321.239,A -85,B 0,C 180,E1 -7584.889,E2 -7584.889} C_VEL
LIN {X 0,Y 467.557,Z 321.245,A -85,B 0,C 180,E1 -7587.773,E2 -7587.773} C_VEL
LIN {X 0,Y 467.562,Z 321.245,A -85,B 0,C 180,E1 -7591.045,E2 -7591.045} C_VEL
LIN {X 0,Y 467.587,Z 321.241,A -85,B 0,C 180,E1 -7594.243,E2 -7594.243} C_VEL
LIN {X 0,Y 467.547,Z 321.246,A -85,B 0,C 180,E1 -7597.187,E2 -7597.187} C_VEL
LIN {X 0,Y 467.554,Z 321.241,A -85,B 0,C 180,E1 -7600.267,E2 -7600.267} C_VEL
LIN {X 0,Y 467.542,Z 321.245,A -85,B 0,C 180,E1 -7603.746,E2 -7603.746} C_VEL
LIN {X 0,Y 467.553,Z 321.248,A -85,B 0,C 180,E1 -7606.256,E2 -7606.256} C_VEL
LIN {X 0,Y 467.578,Z 321.242,A -85,B 0,C 180,E1 -7608.724,E2 -7608.724} C_VEL
LIN {X 0,Y 467.62,Z 321.381,A -85,B 0,C 180,E1 -7610.859,E2 -7610.859} C_VEL
LIN {X 0,Y 468.483,Z 326.941,A -85,B 0,C 180,E1 -7613.652,E2 -7613.652} C_VEL
LIN {X 0,Y 468.537,Z 331.04,A -85,B 0,C 180,E1 -7615.588,E2 -7615.588} C_VEL
LIN {X 0,Y 468.242,Z 338.202,A -85,B 0,C 180,E1 -7618.819,E2 -7618.819} C_VEL
LIN {X 0,Y 468.002,Z 344.96,A -85,B 0,C 180,E1 -7621.769,E2 -7621.769} C_VEL
LIN {X 0,Y 467.67,Z 352.842,A -85,B 0,C 180,E1 -7625.117,E2 -7625.117} C_VEL
LIN {X 0,Y 467.469,Z 359.66,A -85,B 0,C 180,E1 -7627.923,E2 -7627.923} C_VEL
LIN {X 0,Y 467.308,Z 366.48,A -85,B 0,C 180,E1 -7630.679,E2 -7630.679} C_VEL
